ACTION ACT_AXIS:
MC_POWER(
	Axis:=REF , 
	Enable:=power_do , 
	Enable_Positive:=TRUE , 
	Enable_Negative:=TRUE , 
	Override:= , 
	BufferMode:= , 
	Options:= , 
	Status=> , 
	Busy=> , 
	Active=> , 
	Error=> , 
	ErrorID=> );
MC_Read(
	Axis:=REF , 
	Enable:=TRUE , 
	Valid=> , 
	Busy=> , 
	Error=> , 
	ErrorID=> Axis_ErrorId, 
	ErrorStop=> , 
	Disabled=> , 
	Stopping=> , 
	StandStill=> , 
	DiscreteMotion=> , 
	ContinuousMotion=> , 
	SynchronizedMotion=> , 
	Homing=> , 
	ConstantVelocity=> , 
	Accelerating=> , 
	Decelerating=> , 
	Status=> );

MC_Stop(
	Axis:=REF , 
	Execute:=stop_do , 
	Deceleration:= , 
	Jerk:= , 
	Options:= , 
	Done=> , 
	Busy=> , 
	Active=> , 
	CommandAborted=> , 
	Error=> , 
	ErrorID=> );
	IF MC_Stop.Busy THEN 
		stop_do:=FALSE;
	END_IF
MC_Reset(
	Axis:=REF , 
	Execute:=reset_do , 
	Done=> , 
	Busy=> , 
	Error=> , 
	ErrorID=> );
	IF MC_Reset.Busy THEN 
		reset_do:=FALSE;
	END_IF
MC_SetPos(
	Axis:=REF , 
	Execute:=Initialize , 
	Position:=0 , 
	Mode:= , 
	Options:= , 
	Done=> , 
	Busy=> , 
	Error=> , 
	ErrorID=> );
mc_Torque(
	Axis:= REF, 
	Execute:=var_bTorqueCtrlExecute , 
	Relative:= , 
	Torque:=var_rTorque , 
	TorqueRamp:=var_rTorqueRamp , 
	VelocityLimitHigh:= , 
	VelocityLimitLow:= , 
	BufferMode:= , 
	Options:= , 
	InTorque=> , 
	Busy=> , 
	Active=> , 
	CommandAborted=> , 
	Error=> , 
	ErrorId=> );
    IF mc_Torque.Busy THEN 
		var_bTorqueCtrlExecute:=FALSE;
	END_IF
END_ACTION

END_FUNCTION_BLOCK

// ---- POUs/100_SubTank/FB/FB_Circulation.TcPOU
FUNCTION_BLOCK FB_Circulation
VAR_INPUT	
	BottomLevel1,BottomLevel2	:BOOL;	
	MUstate						:INT;
	setoff						:BOOL;
	set_pump_voltage1			:LREAL;
	set_pump_voltage2			:LREAL;
END_VAR
VAR_OUTPUT
	CircPumpWorking1			:BOOL;
	CircPumpWorking2			:BOOL;
	error_code					:INT;
	out_pump_voltage1			:INT;
	out_pump_voltage2			:INT;
END_VAR
VAR
	Bottom_ON_filterTon1		:TON;				//滤波
	Bottom_OFF_filterTon1		:TON;
	Bottom_filterLevel1			:BOOL;
	
	Bottom_ON_filterTon2		:TON;				//滤波
	Bottom_OFF_filterTon2		:TON;
	Bottom_filterLevel2			:BOOL;
	
	filterTime_ON				:TIME;	//接通滤波时间
	filterTime_OFF				:TIME;	//接断开滤波间
	
	ton_circ1,ton_circ2:TON;
	work_ton1,work_ton2:TON;
	circ_time_trig1,circ_time_trig2:R_TRIG;
	circ_number1,circ_number2:INT;//循坏次数
	setoff_f_trig:F_TRIG;
	step_L,step_R:INT;
	state_change_trig1,state_change_trig2:R_TRIG;
	
	EL4002_CH			:ARRAY[1..2] OF FB_WriteAnalog;
	temp_pump_voltage1  :INT;
	temp_pump_voltage2  :INT;
	
END_VAR

ACT_filter_level();
ACT_circ_L();
ACT_circ_R();

IF MUstate=MUStateEnum.swapping THEN 
	filterTime_ON:=T#0S;
	filterTime_OFF:=T#0S;
ELSE
	filterTime_ON:=T#0.5S;
	filterTime_OFF:=T#0.5S;
END_IF

(************setoff***************************)
setoff_f_trig(CLK:=setoff  , Q=> );
IF setoff_f_trig.Q THEN 
	ton_circ1(IN:=FALSE);
	work_ton1(IN:=FALSE);
	ton_circ2(IN:=FALSE);
	work_ton2(IN:=FALSE);
	circ_number1:=0;	
	circ_number2:=0;	
END_IF
(************切换到SWAP或者到idle 时，需将错误复位掉*************************** 2023.1.15 无需复位
state_change_trig1(CLK:=MUstate=MUStateEnum.swapping  , Q=> );
state_change_trig2(CLK:=MUstate=MUStateEnum.idle , Q=> );
IF  state_change_trig1.Q OR state_change_trig2.Q  THEN 
		error_code:=MUErrorEnum.no_error;
		ton_circ1(IN:=FALSE);
		work_ton1(IN:=FALSE);
		ton_circ2(IN:=FALSE);
		work_ton2(IN:=FALSE);
		step_L:=step_R:=0;
END_IF
*)
(**************PUMP  SPEED********************************)
EL4002_CH[1](
	Enable:=TRUE , 
	In:=set_pump_voltage1 , 
	AnalogOffset:= , 
	Set_MaxValue:=5 , 
	MaxValue:=10 , 
	out=>temp_pump_voltage1 );
EL4002_CH[2](
	Enable:=TRUE , 
	In:=set_pump_voltage2 , 
	AnalogOffset:= , 
	Set_MaxValue:=5 , 
	MaxValue:=10 , 
	out=>temp_pump_voltage2 );

IF CircPumpWorking1 THEN 
	out_pump_voltage1:=temp_pump_voltage1;
ELSE
	out_pump_voltage1:=0;
END_IF
IF CircPumpWorking2 THEN 
	out_pump_voltage2:=temp_pump_voltage2;
ELSE
	out_pump_voltage2:=0;
END_IF

ACTION ACT_circ_L:
CASE step_L  OF 
0://
	IF MUstate=MUStateEnum.swapping THEN 
		step_L:=10;
	ELSE
		step_L:=20;
	END_IF
10://swappingg,循坏，不会报错
	IF MUstate<>MUStateEnum.swapping THEN 
		step_L:=20;
	END_IF
	
	CircPumpWorking1:=Bottom_filterLevel1 ;
20://normal,有报错
(*When pump 3 was activate less than …x/min => Alarm 1: Check circulation Left Print Heads
When pump 6 was activate less than …x/min => Alarm 2: Check circulation Right Print Heads

When pump 3 was activate less than 1x/2min =>	Alarm 3: No Circulation through Left Print Heads
When pump 6 was activate less than 1x/2min => 	Alarm 4: No Circulation through Right Print Heads

When pump 3 runs longer than 8sec => 	Alarm 5: Runtime Error Left Circulation pump 
When pump 6 runs longer than 8sec => 	Alarm 6: Runtime Error Right Circulation Pump 

*)
	IF MUstate=MUStateEnum.swapping THEN 
		step_L:=10;
	END_IF
	
	CircPumpWorking1:=Bottom_filterLevel1 ;
	
		ton_circ1(IN:=NOT ton_circ1.Q  , PT:=T#2M , Q=> , ET=> );
		circ_time_trig1(CLK:=CircPumpWorking1 , Q=> );
		IF circ_time_trig1.Q THEN 
				circ_number1:=circ_number1+1;
		END_IF
		
	(*************error********************)
	IF ton_circ1.ET >=T#1M AND ton_circ1.ET<T#2M THEN 				
		IF circ_number1<1 THEN 
			error_code:=MUErrorEnum.alarm_circulation_left;			
		END_IF
	ELSIF ton_circ1.q THEN 		
		IF circ_number1<1 THEN 
			error_code:=MUErrorEnum.alarm_through_left;
		END_IF
		(********error跳转********)
		IF error_code<>0 THEN 
			step_L:=100;
		END_IF
		circ_number1:=0;	
	END_IF
	
	work_ton1(IN:=CircPumpWorking1 , PT:=T#8S , Q=> , ET=> );
	IF work_ton1.Q THEN 
		error_code:=MUErrorEnum.alarm_runtime_circulation_left;	
		step_L:=100;
	END_IF
			
100://error
	CircPumpWorking1:=FALSE;
	circ_number1:=0;	
	ton_circ1(IN:=FALSE);
	work_ton1(IN:=FALSE);
	step_L:=0;

END_CASE
	IF 	setoff    THEN 
		error_code:=MUErrorEnum.no_error;
		step_L:=0;
	END_IF
END_ACTION

ACTION ACT_circ_R:
CASE step_R  OF 
0://
	IF MUstate=MUStateEnum.swapping THEN 
		step_R:=10;
	ELSE
		step_R:=20;
	END_IF
10://swappingg,循坏，不会报错
	IF MUstate<>MUStateEnum.swapping THEN 
		step_R:=20;
	END_IF
	
	CircPumpWorking2:=Bottom_filterLevel2 ;
20://normal,有报错
(*When pump 3 was activate less than …x/min => Alarm 1: Check circulation Left Print Heads
When pump 6 was activate less than …x/min => Alarm 2: Check circulation Right Print Heads

When pump 3 was activate less than 1x/2min =>	Alarm 3: No Circulation through Left Print Heads
When pump 6 was activate less than 1x/2min => 	Alarm 4: No Circulation through Right Print Heads

When pump 3 runs longer than 8sec => 	Alarm 5: Runtime Error Left Circulation pump 
When pump 6 runs longer than 8sec => 	Alarm 6: Runtime Error Right Circulation Pump 

*)
	IF MUstate=MUStateEnum.swapping THEN 
		step_R:=10;
	END_IF
	
	CircPumpWorking2:=Bottom_filterLevel2 ;
	
		ton_circ2(IN:=NOT ton_circ2.Q  , PT:=T#2M , Q=> , ET=> );
		circ_time_trig2(CLK:=CircPumpWorking2 , Q=> );
		IF circ_time_trig2.Q THEN 
				circ_number2:=circ_number2+1;
		END_IF
		
	(*************error********************)
	IF ton_circ2.ET >=T#1M AND ton_circ2.ET<T#2M THEN 				
		IF circ_number2<1 THEN 
			error_code:=MUErrorEnum.alarm_circulation_right;
		END_IF
	ELSIF ton_circ2.q THEN 
		IF circ_number2<1 THEN 
			error_code:=MUErrorEnum.alarm_through_right;
		END_IF
		(********error跳转********)
		IF error_code<>0 THEN 
			step_R:=100;
		END_IF
		circ_number2:=0;	
	END_IF
	
	work_ton2(IN:=CircPumpWorking2 , PT:=T#8S , Q=> , ET=> );
	IF work_ton2.Q THEN 
		error_code:=MUErrorEnum.alarm_runtime_circulation_right;
		step_R:=100;
	END_IF
				
100://error
	CircPumpWorking2:=FALSE;
	circ_number2:=0;	
	ton_circ2(IN:=FALSE);
	work_ton2(IN:=FALSE);
	step_R:=0;

	
END_CASE
	IF setoff   THEN 
		error_code:=MUErrorEnum.no_error;
		step_R:=0;
	END_IF
END_ACTION

ACTION ACT_filter_level:
(************LEVEL_BOT1*****************)
Bottom_ON_filterTon1(IN:=BottomLevel1 , PT:=filterTime_ON , Q=> , ET=> );
Bottom_OFF_filterTon1(IN:=NOT BottomLevel1 , PT:=filterTime_OFF , Q=> , ET=> );

IF Bottom_ON_filterTon1 .Q  THEN 
	Bottom_filterLevel1:=TRUE;
ELSIF Bottom_OFF_filterTon1 .Q THEN 
	Bottom_filterLevel1:=FALSE;
END_IF


(************LEVEL_BOT2*****************)
Bottom_ON_filterTon2(IN:=BottomLevel2 , PT:=filterTime_ON , Q=> , ET=> );
Bottom_OFF_filterTon2(IN:=NOT BottomLevel2 , PT:=filterTime_OFF , Q=> , ET=> );

IF Bottom_ON_filterTon2 .Q  THEN 
	Bottom_filterLevel2:=TRUE;
ELSIF Bottom_OFF_filterTon2 .Q THEN 
	Bottom_filterLevel2:=FALSE;
END_IF
END_ACTION

END_FUNCTION_BLOCK

// ---- POUs/100_SubTank/FB/FB_SubTank_C.TcPOU
FUNCTION_BLOCK FB_SubTank_C
VAR_INPUT	
	sublevel					:BOOL;
	protectLevel				:BOOL;	
	filterTime_ON				:TIME;	//接通滤波时间
	filterTime_OFF				:TIME;	//接断开滤波间
	inkFillTimeOutSet			:TIME;   //供墨超时时间设定 s	
END_VAR
VAR_OUTPUT	
	PumpWorking 				:BOOL;	//输出
	state								:INT;
	error_code					:INT;
	Error						:BOOL;
END_VAR
VAR	
	step						:INT;
	ON_filterTon			:TON;						//滤波
	OFF_filterTon			:TON;
	ON_filterTon_P			:TON;						//保护气瓶滤波
	OFF_filterTon_P			:TON;
	filterLevel			    :BOOL;
	filterLevel_P			:BOOL;
	inkFillTimeOutTon		:TON;	
END_VAR
VAR_IN_OUT
	setoff					:BOOL;
END_VAR

ACT_filter_level();

CASE step OF
0://ready
	state:=SubTankStateEnum.ready;
	(************Pumping*****************)
	IF NOT filterLevel AND NOT filterLevel_P  THEN 		
		PumpWorking :=TRUE;
	END_IF	
	IF 	 filterLevel OR  filterLevel_P  THEN
		PumpWorking :=FALSE;
	END_IF
	
	(************inkFillTimeOut*****************)
	inkFillTimeOutTon(IN:=PumpWorking   , PT:=inkFillTimeOutSet , Q=> , ET=> );
		IF inkFillTimeOutTon.Q THEN 
			error_code:=SubTankErrorEnum.pump_timeout;
			step:=100;	
		END_IF	
	
90://setoff
	error:=FALSE;	
	error_code:=ISSErrorEnum.no_error;
		
	inkFillTimeOutTon(IN:=FALSE);
	PumpWorking  :=FALSE;		
	step:=0;		
	
100://error
	state:=SubTankStateEnum.error;
	inkFillTimeOutTon(IN:=FALSE);
	PumpWorking  :=FALSE;	
	error:=TRUE;
END_CASE

IF setoff OR GVL.Reset THEN 
	setoff:=FALSE;
	step:=90;
END_IF
(*****************************************************)
	IF GVL.Emstop_Button  THEN 
		error_code:=ISSErrorEnum.emergency_error;
		step:=100;
	ELSIF filterLevel_P THEN 
		error_code:=ISSErrorEnum.back_to_air_tank;
		step:=100;
	END_IF

ACTION ACT_filter_level:
(************LEVEL*****************)
ON_filterTon(IN:=sublevel , PT:=filterTime_ON , Q=> , ET=> );
OFF_filterTon(IN:=NOT sublevel , PT:=filterTime_OFF , Q=> , ET=> );

IF ON_filterTon .Q  THEN 
	filterLevel:=TRUE;
ELSIF OFF_filterTon .Q THEN 
	filterLevel:=FALSE;
END_IF

(*************LEVEL_P****************)
ON_filterTon_P(IN:=protectLevel , PT:=filterTime_ON , Q=> , ET=> );
OFF_filterTon_P(IN:=NOT protectLevel , PT:=filterTime_OFF , Q=> , ET=> );

IF ON_filterTon_P .Q  THEN 
	filterLevel_P:=TRUE;
ELSIF OFF_filterTon_P .Q THEN 
	filterLevel_P:=FALSE;
END_IF
END_ACTION

END_FUNCTION_BLOCK

// ---- POUs/100_SubTank/FB/FB_SubTank_W.TcPOU
FUNCTION_BLOCK FB_SubTank_W
VAR_INPUT
	enable							:BOOL;
	fill_in_swap_enable				:BOOL;
	ISswappingState					:INT;//是否在换液状态
	alternate_fill					:BOOL;//交替加墨
	Toplevel          				:BOOL;
	protectLevel					:BOOL;	
	filterTime_ON					:TIME;	//接通滤波时间
	filterTime_OFF					:TIME;	//接断开滤波间
	inkFillTimeOutSet				:TIME;   //供墨超时时间设定 s	
	CircPumpWorking			        :BOOL;
END_VAR
VAR_OUTPUT	
	PumpWorking				    :BOOL;	//输出	
	state						:INT;
	error_code					:INT;
	Error						:BOOL;
END_VAR
VAR	
	step1,step2,step						:INT;
	Top_ON_filterTon				:TON;					//滤波
	Top_OFF_filterTon				:TON;
	Top_filterLevel					:BOOL;
	inkFillTimeOutTon				:TON;
	
	ON_filterTon_P			:TON;						//滤波
	OFF_filterTon_P			:TON;
	filterLevel_P				:BOOL;
	en_r_trig:R_TRIG;
	en_f_trig:F_TRIG;
	FB_SQUARE			:FB_SQUARE;
	ton1:Tc2_Standard.TON;
END_VAR
VAR_IN_OUT
	setoff					:BOOL;
END_VAR

ACT_fill();


	IF   GVL.Emstop_Button THEN 
		error_code:=ISSErrorEnum.emergency_error;
		step:=100;	
	
	ELSIF filterLevel_P THEN 
		error_code:=ISSErrorEnum.back_to_air_tank;
		step:=100;
	END_IF

ACTION ACT_fill:
ACT_filter_level();
(******************FillPumpWorking********************)
CASE step OF
0://ready
	state:=SubTankStateEnum.ready;
	
(********************供墨*************************************************************************************)	
	(************setoff*****************)	
	IF setoff OR GVL.Reset THEN 
		step:=90;
	END_IF
	IF enable THEN 
		IF ISswappingState<>MUStateEnum.swapping THEN  //正常供墨
			ACT_fill_in_normal();
		ELSE 											//交换加墨	
			ACT_fill_in_swap();
		END_IF	
	ELSE 
		inkFillTimeOutTon(IN:=FALSE);
		PumpWorking :=FALSE;
	END_IF			
90://setoff
		error:=FALSE;	
		error_code:=ISSErrorEnum.no_error;
		
		inkFillTimeOutTon(IN:=FALSE);
		PumpWorking :=FALSE;	
		step:=0;
100://error
	state:=ISSStateEnum.error;
	inkFillTimeOutTon(IN:=FALSE);
	PumpWorking :=FALSE;	
	error:=TRUE;	
END_CASE

IF setoff OR GVL.Reset THEN 
	setoff:=FALSE;
	step:=90;
END_IF
END_ACTION

ACTION ACT_fill_in_normal:
ACT_filter_level();
(******************FillPumpWorking********************)
	(************Pumping*****************)
	IF NOT filterLevel_P  AND  NOT Top_filterLevel  AND NOT CircPumpWorking THEN 
		PumpWorking:=TRUE;
	END_IF	
	IF 	 filterLevel_P  OR Top_filterLevel  OR CircPumpWorking THEN 
		PumpWorking:=FALSE;
	END_IF
	

	(************inkFillTimeOut*****************)
		inkFillTimeOutTon(IN:=PumpWorking  , PT:=inkFillTimeOutSet, Q=> , ET=> );
		IF inkFillTimeOutTon.Q THEN 
			error_code:=SubTankErrorEnum.pump_timeout;
			step:=100;	
		END_IF
END_ACTION

ACTION ACT_fill_in_swap:
en_r_trig(CLK:= fill_in_swap_enable, Q=> );
en_f_trig(CLK:=fill_in_swap_enable , Q=> );
IF en_r_trig.Q  OR en_f_trig .Q  THEN 
		PumpWorking  :=FALSE;				
		inkFillTimeOutTon(IN:=FALSE);
END_IF
(******************FillPumpWorking********************)
IF fill_in_swap_enable THEN 
		IF NOT alternate_fill THEN 
				(************all Pumping*****************)
			IF NOT filterLevel_P  AND  NOT Toplevel  AND NOT CircPumpWorking THEN 
				PumpWorking:=TRUE;
			END_IF	
			IF 	 filterLevel_P  OR Toplevel  OR CircPumpWorking THEN 
				PumpWorking:=FALSE;
			END_IF
				
			(************inkFillTimeOut*****************)
				inkFillTimeOutTon(IN:=PumpWorking  , PT:=T#2M, Q=> , ET=> );				
				IF inkFillTimeOutTon.Q THEN 
					error_code:=SubTankErrorEnum.pump_timeout;
					step:=100;			
				END_IF	
		ELSE
				(************alternate Pumping*****************)		
			IF NOT filterLevel_P  AND  NOT Toplevel  AND NOT CircPumpWorking THEN
				FB_SQUARE(T_ON:=T[2] , T_OFF:= T[3], SQUARE=> PumpWorking); 
				inkFillTimeOutTon(IN:=TRUE  , PT:=T#2M, Q=> , ET=> );
				IF inkFillTimeOutTon.Q THEN 
					error_code:=SubTankErrorEnum.pump_timeout;
					step:=100;
				END_IF
			END_IF	
			IF 	 filterLevel_P  OR Toplevel  OR CircPumpWorking THEN 
				PumpWorking:=FALSE;		
			END_IF
			
		END_IF
END_IF
END_ACTION

ACTION ACT_filter_level:
(************LEVEL_TOP*****************)
Top_ON_filterTon(IN:=Toplevel , PT:=filterTime_ON , Q=> , ET=> );
Top_OFF_filterTon(IN:=NOT Toplevel , PT:=filterTime_OFF , Q=> , ET=> );

IF Top_ON_filterTon .Q  THEN 
	Top_filterLevel:=TRUE;
ELSIF Top_OFF_filterTon .Q THEN 
	Top_filterLevel:=FALSE;
END_IF



(************LEVEL_P*****************)
ON_filterTon_P(IN:=protectLevel , PT:=filterTime_ON-T#1S , Q=> , ET=> );
OFF_filterTon_P(IN:=NOT protectLevel , PT:=filterTime_OFF-T#1S , Q=> , ET=> );

IF ON_filterTon_P .Q  THEN 
	filterLevel_P:=TRUE;
ELSIF OFF_filterTon_P .Q THEN 
	filterLevel_P:=FALSE;
END_IF
END_ACTION

END_FUNCTION_BLOCK

// ---- POUs/100_SubTank/P_SubTank.TcPOU
PROGRAM P_SubTank
VAR
	FB_SubTankFill_C   :ARRAY[1..12] OF FB_SubTank_C;
	FB_SubTankFill_P   :ARRAY[1..2] OF FB_SubTank_C;
	FB_SubTankFill_W   :ARRAY[1..2] OF FB_SubTank_W;
	FB_SubTankFill_F   :ARRAY[1..2] OF FB_SubTank_W;
	
	PumpWorking1_W,PumpWorking2_W:BOOL;
	PumpWorking1_F,PumpWorking2_F:BOOL;
	
	bqFillPumpWorking_W_r_trig:Tc2_Standard.R_TRIG;//白墨泵启动
	bqFillPumpWorking_F_r_trig:Tc2_Standard.R_TRIG;	//	清洗液泵启动
	
	i:INT;
(****************白墨循坏*******************************)
	FB_Circulation:FB_Circulation;
	
	enable_W_rtrig:Tc2_Standard.R_TRIG;
	enable_F_rtrig:Tc2_Standard.R_TRIG;
END_VAR

VAR PERSISTENT
	SubTankFill_en:ARRAY[1..4] OF BOOL:=[1,1,0,0];//w1,w2,f1,f2  白，清洗液供墨使能
END_VAR

ACT_Color();
ACT_W_F();
ACT_Circulation();
(****white pump**************************************)
stOutput.bqFillPumpWorking[13]:=(PumpWorking1_W ) 
						AND NOT stOutput.bqFillPumpWorking[19] ;
stOutput.bqFillPumpWorking[15]:=(PumpWorking2_W ) 
						AND NOT stOutput.bqFillPumpWorking[20];
(****flush pump**************************************)
stOutput.bqFillPumpWorking[19]:=(PumpWorking1_F ) 
						AND NOT stOutput.bqFillPumpWorking[13] ;
stOutput.bqFillPumpWorking[20]:=(PumpWorking2_F ) 
						AND NOT stOutput.bqFillPumpWorking[15] ;
													
(**********************墨盒里 
		0” circuit not filled (default setting)
	“1” circuit filled with “white ink”
	“2” circuit filled with “storage fluid”
******************************************************)
bqFillPumpWorking_W_r_trig(CLK:=stOutput.bqFillPumpWorking[13] OR stOutput.bqFillPumpWorking[15] , Q=> );
bqFillPumpWorking_F_r_trig(CLK:=stOutput.bqFillPumpWorking[19] OR stOutput.bqFillPumpWorking[20] , Q=> );
IF bqFillPumpWorking_W_r_trig.Q THEN
	SubTankInk_type:=1; 
ELSIF bqFillPumpWorking_F_r_trig.Q THEN 
	SubTankInk_type:=2;
END_IF


(***************切换墨水**************************)
enable_F_rtrig(CLK:= GVL_API.stMU.state=MUStateEnum.swapping AND GVL_API.stMU.cycle=0 , Q=> );
enable_W_rtrig(CLK:=GVL_API.stMU.state=MUStateEnum.swapping AND GVL_API.stMU.cycle=1 , Q=> );
IF enable_W_rtrig.Q THEN  //WHITE
	SubTankFill_en[1]:=TRUE;
	SubTankFill_en[2]:=TRUE;
	SubTankFill_en[3]:=FALSE;
	SubTankFill_en[4]:=FALSE;
ELSIF enable_F_rtrig.Q THEN //FLUSH
	SubTankFill_en[1]:=FALSE;
	SubTankFill_en[2]:=FALSE;
	SubTankFill_en[3]:=TRUE;
	SubTankFill_en[4]:=TRUE;
END_IF

ACTION ACT_Circulation:
FB_Circulation(
	BottomLevel1:=GVL.inklevel_W_L_BOT , 
	BottomLevel2:=GVL.inklevel_W_R_BOT , 
	MUstate:=GVL_API.stMU.state , 
	setoff:= GVL_API.stMU.SetOff OR GVL.Reset, 
	set_pump_voltage1:=HMI_CircPump1_V , 
	set_pump_voltage2:=HMI_CircPump2_V , 
	CircPumpWorking1=>stOutput.bqSubCircPumpWorking[1]  , 
	CircPumpWorking2=> stOutput.bqSubCircPumpWorking[2] , 
	error_code=> ,
	out_pump_voltage1=>EL4002_S[1] , 
	out_pump_voltage2=>EL4002_S[2] );
END_ACTION

ACTION ACT_Color:
(*******************COLOR***************************)
(*
1	:	LC1		2	:	LC2
3	:	LM1		4	:	LM2
5	:	Y1		6	:	Y2
7	:	M1		8	:	M2
9	:	C1		10	:	C2
11	:	K1		12	:	K2
13		P1		14		P2
15		W_L		16		W_R

*)
FOR i:=1 TO 12 DO 
	FB_SubTankFill_C[i](
		sublevel:= stInput.biSubInkTankLevel[i], 
		protectLevel:= stInput.biProtectAirTankLevel_C, 
		filterTime_ON:= T#0S, 
		filterTime_OFF:= T#3S, 
		inkFillTimeOutSet:= LREAL_TO_TIME(GVL_API.stSubTank[i].timeout) ,
		PumpWorking=> stOutput.bqFillPumpWorking[i], 
		state=> GVL_API.stSubTank[i].state, 
		error_code=> GVL_API.stSubTank[i].error_code, 
		Error=> GVL_API.stSubTank[i].Error, 
		setoff:=GVL_API.stSubTank[i].Setoff );
END_FOR

(*******************Primer***************************)
	FB_SubTankFill_P[1](
		sublevel:= stInput.biSubInkTankLevel[17], 
		protectLevel:= stInput.biProtectAirTankLevel_W, 
		filterTime_ON:= T#0S, 
		filterTime_OFF:= T#3S, 
		inkFillTimeOutSet:= LREAL_TO_TIME(GVL_API.stSubTank[13].timeout), 
		PumpWorking=> stOutput.bqFillPumpWorking[17], 
		state=> GVL_API.stSubTank[13].state, 
		error_code=> GVL_API.stSubTank[13].error_code, 
		Error=> GVL_API.stSubTank[13].Error, 
		setoff:=GVL_API.stSubTank[13].Setoff );
	FB_SubTankFill_P[2](
		sublevel:= stInput.biSubInkTankLevel[18], 
		protectLevel:= stInput.biProtectAirTankLevel_W, 
		filterTime_ON:= T#0S, 
		filterTime_OFF:= T#3S, 
		inkFillTimeOutSet:= LREAL_TO_TIME(GVL_API.stSubTank[14].timeout), 
		PumpWorking=> stOutput.bqFillPumpWorking[18], 
		state=> GVL_API.stSubTank[14].state, 
		error_code=> GVL_API.stSubTank[14].error_code, 
		Error=> GVL_API.stSubTank[14].Error, 
		setoff:=GVL_API.stSubTank[14].Setoff );
END_ACTION

ACTION ACT_W_F:
(*******************WHITE/FLUSH***************************)	
GVL.inklevel_W_L_BOT:=stInput.biSubInkTankLevel[13] ;	//W_L_BOT
GVL.inklevel_W_L_TOP:=stInput.biSubInkTankLevel[14] ;	//W_L_TOP
GVL.inklevel_W_R_TOP:=stInput.biSubInkTankLevel[15] ;	//W_R_TOP
GVL.inklevel_W_R_BOT:=stInput.biSubInkTankLevel[16] ;	//W_R_BOT


(*******************white***************************)
	FB_SubTankFill_W[1](
		enable:=SubTankFill_en[1],
		fill_in_swap_enable:=GVL.fill_W_in_swap_enable , 
		ISswappingState:=GVL_API.stMU.state  , 
		alternate_fill:= P_MaintenanceUnit.FB_Auto_Cycles_Swap.alternate_Pumping, 
		Toplevel:= GVL.inklevel_W_L_TOP, 
		protectLevel:= stInput.biProtectAirTankLevel_W, 
		filterTime_ON:= T#0S, 
		filterTime_OFF:= T#3S, 
		inkFillTimeOutSet:= inkFillTimeOutSet, 
		CircPumpWorking:= stOutput.bqSubCircPumpWorking[1], 
		PumpWorking=> PumpWorking1_W, 
		state=> GVL_API.stSubTank[15].state, 
		error_code=> GVL_API.stSubTank[15].error_code, 
		Error=> GVL_API.stSubTank[15].Error, 
		setoff:= GVL_API.stSubTank[15].Setoff);
	FB_SubTankFill_W[2](
		enable:=SubTankFill_en[2],
		fill_in_swap_enable:=GVL.fill_W_in_swap_enable , 
		ISswappingState:=GVL_API.stMU.state  , 
		alternate_fill:= P_MaintenanceUnit.FB_Auto_Cycles_Swap.alternate_Pumping, 
		Toplevel:= GVL.inkLevel_W_R_TOP, 
		protectLevel:= stInput.biProtectAirTankLevel_W, 
		filterTime_ON:= T#0S, 
		filterTime_OFF:= T#3S, 
		inkFillTimeOutSet:= inkFillTimeOutSet, 
		CircPumpWorking:= stOutput.bqSubCircPumpWorking[2], 
		PumpWorking=> PumpWorking2_W, 
		state=> GVL_API.stSubTank[16].state, 
		error_code=> GVL_API.stSubTank[16].error_code, 
		Error=> GVL_API.stSubTank[16].Error, 
		setoff:= GVL_API.stSubTank[16].Setoff);	
		
(*******************FLUSH***************************)
	FB_SubTankFill_F[1](
		enable:=SubTankFill_en[3],
		fill_in_swap_enable:=GVL.fill_F_in_swap_enable , 
		ISswappingState:=GVL_API.stMU.state  , 
		alternate_fill:= P_MaintenanceUnit.FB_Auto_Cycles_Swap.alternate_Pumping, 
		Toplevel:= GVL.inklevel_W_L_TOP, 
		protectLevel:= stInput.biProtectAirTankLevel_W, 
		filterTime_ON:= T#0S, 
		filterTime_OFF:= T#3S, 
		inkFillTimeOutSet:= inkFillTimeOutSet, 
		CircPumpWorking:= stOutput.bqSubCircPumpWorking[1], 
		PumpWorking=> PumpWorking1_F, 
		state=> GVL_API.stSubTank[15].state, 
		error_code=> GVL_API.stSubTank[15].error_code, 
		Error=> GVL_API.stSubTank[15].Error, 
		setoff:= GVL_API.stSubTank[15].Setoff);
	FB_SubTankFill_F[2](
		enable:=SubTankFill_en[4],
		fill_in_swap_enable:=GVL.fill_F_in_swap_enable , 
		ISswappingState:=GVL_API.stMU.state  , 
		alternate_fill:= P_MaintenanceUnit.FB_Auto_Cycles_Swap.alternate_Pumping, 
		Toplevel:= GVL.inkLevel_W_R_TOP, 
		protectLevel:= stInput.biProtectAirTankLevel_W, 
		filterTime_ON:= T#0S, 
		filterTime_OFF:= T#3S, 
		inkFillTimeOutSet:= inkFillTimeOutSet, 
		CircPumpWorking:= stOutput.bqSubCircPumpWorking[2], 
		PumpWorking=> PumpWorking2_F, 
		state=> GVL_API.stSubTank[16].state, 
		error_code=> GVL_API.stSubTank[16].error_code, 
		Error=> GVL_API.stSubTank[16].Error, 
		setoff:= GVL_API.stSubTank[16].Setoff);
END_ACTION

END_PROGRAM

// ---- POUs/999_TwinSAFE/P_TwinSAFE.TcPOU
PROGRAM P_TwinSAFE
VAR
	Err_Ack		AT%Q* 	:BOOL;//当出现了通讯报错时，用来做安全应答
	//Run_Stop	AT%Q* 	:BOOL;//启动或停止安全程序运行
	//Restart		AT%Q* 	:BOOL;//重启安全程序
	//Relyback	AT%Q* 	:ARRAY [1..4] OF BOOL;
	
	Com_err		AT%I* 	:BOOL;//用来显示通讯报错
	FB_err		AT%I* 	:BOOL;//用来显示功能块报错
	//FB_run		AT%I* 	:BOOL;
	
(**************FB监控**********************)	
	TwinSAFE_Group_State     					AT%I*    :USINT;
	TwinSAFE_FBstop1_State	 					AT%I*    :USINT;	
	TwinSAFE_Group_State_Enum				:TwinSAFE_Group_State_Enum;
	TwinSAFE_FB_ESTOP_State_Enum			:TwinSAFE_FB_ESTOP_State_Enum;	
	FB_COE_READ									:ARRAY[1..4] OF Tc2_EtherCAT.FB_EcCoESdoRead;
	bCoe_read											:BOOL;
	
(*************接入EL1094***********************)	
	bishuttle_crash_detector_left					:BOOL;
	bishuttle_crash_detector_right					:BOOL;
	btEmergency_stop									:BOOL;
	Emergency_stop_2904									:BOOL;
	biinterlock 			  								:ARRAY[1..8] OF BOOL;
	rely_back  												:ARRAY[1..4] OF BOOL;
	btReset													:BOOL;
	
(*******************LOG*****************)
	i:INT;
	Coe_Read_ton:ton;	
	log_ID:INT;
	last_group_state_ton:Tc2_Standard.TON;
	last_group_state:USINT;
	last_FBstop1_state_ton:Tc2_Standard.TON;
	last_FBstop1_state:USINT;
	
END_VAR

(*
EDM 接收反馈，假如多个的话，反馈用1904 ，可以用FB_ADD，此模块只可以用安全模块输入
不用1904，反馈需在PLC内，就做好合并，以一个值直接传输到TianSAFE 内的变量
*)

ACT_LOG();
ACT_Match();
stInput.btReset:=btReset;
Err_Ack:=stInput.btReset;


Coe_Read_ton(IN:=NOT Coe_Read_ton.Q  , PT:= , Q=> , ET=> );
IF Coe_Read_ton.Q THEN 
	bCoe_read:=NOT bCoe_read;
END_IF
FOR i:=1 TO 4 DO
FB_COE_READ[i](
	sNetId:= '192.168.1.138.2.1'(*'5.88.78.180.2.1'*) , 
	nSlaveAddr:=1014 , 
	nSubIndex:= INT_TO_BYTE(i), 
	nIndex:=16#7001 , 
	pDstBuf:=ADR(EL2904[1,i]) , 
	cbBufLen:=SIZEOF(EL2904[1,i]) , 
	bExecute:= bCoe_read, 
	tTimeout:= , 
	bBusy=> , 
	bError=> , 
	nErrId=> , 
	cbRead=> );
END_FOR

ACTION ACT_LOG:
(*************************LOG*******************************************)
//只记录错误
log_ID:=460;

//Com_err
AlarmActionArray[log_ID+1].AlarmMsg.EN	:=	'TwinSAFE Com_err ';
fbSetAlarm[log_ID+1](
	InUse:=TRUE , 
	//EventId:=log_ID+2 , 
	EventActive:=Com_err , 
	EventClass:=Alm_EventClass.Alarm , 
	ToTheLogFile:=TRUE, 
	ToTheHistory:=TRUE , 
 );
 
 //FB_err
AlarmActionArray[log_ID+2].AlarmMsg.EN	:=	'TwinSAFE FB_err ';
fbSetAlarm[log_ID+2](
	InUse:=TRUE , 
	//EventId:=log_ID+2 , 
	EventActive:=FB_err , 
	EventClass:=Alm_EventClass.Alarm , 
	ToTheLogFile:=TRUE, 
	ToTheHistory:=TRUE , 
 );

  //Restart
AlarmActionArray[log_ID+3].AlarmMsg.EN	:=	'TwinSAFE Restart ';
fbSetAlarm[log_ID+3](
	InUse:=TRUE , 
	//EventId:=log_ID+3 , 
	EventActive:=gvl.Reset , 
	EventClass:=Alm_EventClass.Event , 
	ToTheLogFile:=TRUE, 
	ToTheHistory:=TRUE , 
 );
 
//	TwinSAFE_Group_State
last_group_state_ton(IN:=NOT last_group_state_ton.Q  , PT:=T#200MS , Q=> , ET=> );
IF last_group_state_ton.Q THEN 
	last_group_state:=TwinSAFE_Group_State;
END_IF
CASE TwinSAFE_Group_State OF
1	:	TwinSAFE_Group_State_Enum	:=	1	;
2	:	TwinSAFE_Group_State_Enum	:=	2	;
4	:	TwinSAFE_Group_State_Enum	:=	4	;
5	:	TwinSAFE_Group_State_Enum	:=	5	;
6	:	TwinSAFE_Group_State_Enum	:=	6	;
7	:	TwinSAFE_Group_State_Enum	:=	7	;
16	:	TwinSAFE_Group_State_Enum	:=	16	;
17	:	TwinSAFE_Group_State_Enum	:=	17	;
END_CASE
AlarmActionArray[log_ID+4].AlarmMsg.EN	:=	CONCAT('TwinSAFE_Group_State:',
																	TO_STRING(TwinSAFE_Group_State_Enum));

fbSetAlarm[log_ID+4](
	InUse:=TRUE , 
	//EventId:=log_ID+2 , 
	EventActive:=last_group_state<>TwinSAFE_Group_State , 
	EventClass:=Alm_EventClass.Message , 
	ToTheLogFile:=TRUE, 
	ToTheHistory:=TRUE , 
 );

//TwinSAFE_FBstop1_State
last_FBstop1_state_ton(IN:=NOT last_FBstop1_state_ton.Q  , PT:=T#200MS , Q=> , ET=> );
IF last_FBstop1_state_ton.Q THEN 
	last_FBstop1_state:=TwinSAFE_FBstop1_State;
END_IF

CASE TwinSAFE_FBstop1_State OF
0	:	TwinSAFE_FB_ESTOP_State_Enum	:=	0	;
1	:	TwinSAFE_FB_ESTOP_State_Enum	:=	1	;
2	:	TwinSAFE_FB_ESTOP_State_Enum	:=	2	;
3	:	TwinSAFE_FB_ESTOP_State_Enum	:=	3	;
4	:	TwinSAFE_FB_ESTOP_State_Enum	:=	4	;
5	:	TwinSAFE_FB_ESTOP_State_Enum	:=	5	;
6	:	TwinSAFE_FB_ESTOP_State_Enum	:=	6	;
8	:	TwinSAFE_FB_ESTOP_State_Enum	:=	8	;
END_CASE
AlarmActionArray[log_ID+5].AlarmMsg.EN	:=	CONCAT('TwinSAFE_FBstop1_State:',
																	TO_STRING(TwinSAFE_FB_ESTOP_State_Enum));

fbSetAlarm[log_ID+5](
	InUse:=TRUE , 
	//EventId:=log_ID+2 , 
	EventActive:=last_FBstop1_state<>TwinSAFE_FBstop1_State , 
	EventClass:=Alm_EventClass.Message , 
	ToTheLogFile:=TRUE, 
	ToTheHistory:=TRUE , 
 );
END_ACTION

ACTION ACT_Match:
Emergency_stop_2904						:=(NOT EL2904[1,1] OR NOT EL2904[1,2])  ;
btEmergency_stop					:=NOT EL1904_M[1,1] OR NOT EL1904_M[1,2];

Axis[FastScan].IO.snLimitN			:=EL1904_M[1,3];
Axis[FastScan].IO.snLimitP			:=EL1904_M[1,4];
bishuttle_crash_detector_left		:=EL1904_M[2,1];
bishuttle_crash_detector_right		:=EL1904_M[2,2];
biinterlock[1]								:=EL1904_M[2,3];
biinterlock[2]								:=EL1904_M[2,4];
biinterlock[3]								:=EL1904_M[3,1];
biinterlock[4]								:=EL1904_M[3,2];
biinterlock[5]								:=EL1904_M[3,3];
biinterlock[6]								:=EL1904_M[3,4];
biinterlock[7]								:=EL1904_M[4,1];
biinterlock[8]								:=EL1904_M[4,2];
btReset										:=EL1904_M[4,3];

rely_back[1]								:=EL1904_M[5,1];
rely_back[2]								:=EL1904_M[5,2];
rely_back[3]								:=EL1904_M[5,3];
rely_back[4]								:=EL1904_M[5,4];
END_ACTION

END_PROGRAM

// ---- POUs/040_System/SystemEnvironment/P_SystemEnvironment.TcPOU
PROGRAM P_SystemEnvironment
VAR
	FB_SystemEnvironment:FB_SystemEnvironment;
	i:INT;
	log_ErrorEnum:EnvironmentErrorEnum;
	log_ID:INT;
END_VAR

ACT_LOG();
FB_SystemEnvironment(
	IO_Error:=P_Modbus_RTU.station_error[3] , 
	duration:= GVL_API.stSystemEnvironment.duration, 
	period:=GVL_API.stSystemEnvironment.period , 
	temp_measured=>GVL_API.stSystemEnvironment.temp_measured, 
	humidity_measured=> GVL_API.stSystemEnvironment.humidity_measured, 
	bqbuzzer=>stOutput.bqBuzzer , 
	Error=> GVL_API.stSystemEnvironment.Error, 
	error_code:= GVL_API.stSystemEnvironment.error_code, 
	state:= GVL_API.stSystemEnvironment.state, 
	Reset:=GVL_API.stSystemEnvironment.Reset  ,
	BuzzerOn:=GVL_API.stSystemEnvironment.BuzzerOn,
	BuzzerOff:=GVL_API.stSystemEnvironment.BuzzerOff );

ACTION ACT_LOG:
(*************************LOG*******************************************)
log_ID:=450;

//ERROR,log_ErrorEnum只能等于一个常数,   
CASE GVL_API.stSystemEnvironment.error_code  OF
0	:	log_ErrorEnum	:=	0	;
1	:	log_ErrorEnum	:=	1	;
2	:	log_ErrorEnum	:=	2	;
3	:	log_ErrorEnum	:=	3	;
4	:	log_ErrorEnum	:=	4	;
666	:	log_ErrorEnum	:=	666	;

END_CASE

AlarmActionArray[log_ID+1].AlarmMsg.EN	:=CONCAT('SystemEnvironment Error: ',TO_STRING(log_ErrorEnum));
fbSetAlarm[log_ID+1](
	InUse:=TRUE , 
	EventId:=log_ID+1 , 
	EventActive:=GVL_API.stSystemEnvironment.error_code<>0  AND GVL_API.stSystemEnvironment.error_code<>666, 
	EventClass:=Alm_EventClass.Alarm , 
	ToTheLogFile:=TRUE, 
	ToTheHistory:=TRUE , 
 );
 
//reset
AlarmActionArray[log_ID+2].AlarmMsg.EN	:=	'SystemEnvironment Reset ';
fbSetAlarm[log_ID+2](
	InUse:=TRUE , 
	EventId:=log_ID+2 , 
	EventActive:=GVL_API.stSystemEnvironment.Reset  , 
	EventClass:=Alm_EventClass.Event , 
	ToTheLogFile:=TRUE, 
	ToTheHistory:=TRUE , 
 );
 
 //buzz on
AlarmActionArray[log_ID+3].AlarmMsg.EN	:=CONCAT(('SystemEnvironment BuzzerOn duration: '),
																	LREAL_TO_STRING(GVL_API.stSystemEnvironment.duration));																	
AlarmActionArray[log_ID+3].AlarmMsg.EN	:=CONCAT(AlarmActionArray[log_ID+3].AlarmMsg.EN,', period: ');
AlarmActionArray[log_ID+3].AlarmMsg.EN	:=CONCAT(AlarmActionArray[log_ID+3].AlarmMsg.EN,
																	LREAL_TO_STRING(GVL_API.stSystemEnvironment.period));																															
fbSetAlarm[log_ID+3](
	InUse:=TRUE , 
	EventId:=log_ID+3 , 
	EventActive:=GVL_API.stSystemEnvironment.BuzzerOn  , 
	EventClass:=Alm_EventClass.Event , 
	ToTheLogFile:=TRUE, 
	ToTheHistory:=TRUE , 
 );
 
  //buzz off
AlarmActionArray[log_ID+4].AlarmMsg.EN	:='SystemEnvironment BuzzerOff ';
																													
fbSetAlarm[log_ID+4](
	InUse:=TRUE , 
	EventId:=log_ID+4 , 
	EventActive:= GVL_API.stSystemEnvironment.BuzzerOff  , 
	EventClass:=Alm_EventClass.Event , 
	ToTheLogFile:=TRUE, 
	ToTheHistory:=TRUE , 
 );
END_ACTION

END_PROGRAM

// ---- POUs/090MaintenanceUnit/FB/FB_drip_purge.TcPOU
(*不管什么时候，V7先断，再断V8,V9*)
FUNCTION_BLOCK FB_drip_purge
VAR_INPUT
	start_exe					    :BOOL;
	IntervalTime_W 			:LREAL;//min
	DripTime_W 				:LREAL;//sec
	PurgeTime_W 			:LREAL;//sec
	IntervalTime_C 			:LREAL;//min
	DripTime_C 				:LREAL;//sec
	PurgeTime_C 			   :LREAL;//sec
END_VAR
VAR_OUTPUT
	PurgeValve7				:BOOL;
	VacWhiteValve8			:BOOL;
	VacColorValve9			:BOOL;
	
END_VAR
VAR_IN_OUT
	has_dripped				:BOOL;
END_VAR
VAR
	start_r_trig:R_TRIG;
	start_f_trig:F_TRIG;
	step_change_trig:ARRAY[1..3] OF R_TRIG;
	step_change_en:BOOL;
	enable: BOOL;
	step:INT;
	step_W,step_C:INT;
	

	ton_IntervalTime_W 			:TON;//min
	ton_DripTime_W 				:TON;//sec
	ton_PurgeTime_W 			:TON;//sec
	ton_IntervalTime_C 			:TON;//min
	ton_DripTime_C 				:TON;//sec
	ton_PurgeTime_C 			:TON;//sec
	ton_delay					:TON;
	max_IntervalTime			:LREAL;
	ton_IntervalTime		 	:TON;//min
	
	Need_D_P_White:BOOL;//白墨时间到，需要滴压墨
	Need_D_P_Color:BOOL;//彩墨时间到，需要滴压墨
	step_both:INT;
	
	Dripping_trig:R_TRIG;
END_VAR

start_r_trig(CLK:= start_exe , Q=> );
start_f_trig(CLK:=start_exe , Q=> );

IF start_r_trig.Q THEN
	enable :=TRUE;
	//has_dripped:=FALSE;
END_IF
IF start_f_trig.Q OR GVL.Emstop_Button THEN
	enable :=FALSE;
	//has_dripped:=FALSE;
END_IF


(*切换条件：1：按设置时间；
2:V7,V8,V9停止时
*)
IF NOT PurgeValve7 AND NOT VacWhiteValve8 AND NOT VacColorValve9 THEN 
	step_change_en:=TRUE;
ELSE step_change_en:=FALSE;
END_IF

IF step_change_en THEN 
	IF PurgeTime_W=0  AND PurgeTime_C=0 THEN 
			step:=1;
	ELSIF DripTime_W=0 AND DripTime_C=0 AND PurgeTime_W= PurgeTime_C 
			AND IntervalTime_W=IntervalTime_C THEN 
			step:=2;
	ELSE 
			step:=3;
	END_IF
END_IF
		
CASE step OF
1:ACT_eg1();
2:ACT_eg2();
3:ACT_eg3();
END_CASE

(*Going off means the upper SW is closed
- As soon as the upper SW is restarted we read that value (is should be true if you have dripped)
- Then we  will reset that value en everything restarts all over again
*)
Dripping_trig(CLK:=PurgeValve7 OR VacWhiteValve8 OR VacColorValve9 , Q=> );
IF Dripping_trig.Q THEN 
	has_dripped:=TRUE;
END_IF

ACTION ACT_eg1:
IF enable THEN 
	ton_IntervalTime_W(IN:=NOT ton_IntervalTime_W.Q , PT:=LREAL_TO_TIME(IntervalTime_W)*1000*60 , Q=> , ET=> );
	ton_IntervalTime_C(IN:=NOT ton_IntervalTime_C.Q , PT:=LREAL_TO_TIME(IntervalTime_C)*1000*60 , Q=> , ET=> );
ELSE 
	ton_IntervalTime_W(IN:=FALSE);
	ton_IntervalTime_C(IN:=FALSE);
	ton_DripTime_W(IN:=FALSE);
	ton_DripTime_C(IN:=FALSE);
	step_W:=0;
	step_C:=0;	
	VacWhiteValve8:=FALSE;
	VacColorValve9:=FALSE;
	
END_IF
(******************Drip_White*****************************)
CASE step_W OF 
0://间隔
	IF ton_IntervalTime_W.Q THEN 
		step_W:=10;
	END_IF
10:
	IF DripTime_W>0 THEN 
		step_W:=20;
	ELSE 
		step_W:=0;
	END_IF
20:
	ton_DripTime_W(IN:=TRUE , PT:=LREAL_TO_TIME(DripTime_W)*1000 , Q=> , ET=> );
	VacWhiteValve8:=TRUE;
	IF ton_DripTime_W.Q THEN 
		step_W:=30;
	END_IF
30:
	VacWhiteValve8:=FALSE;
	ton_DripTime_W(IN:=FALSE);
	step_W:=0;
END_CASE
(******************Drip_Color*****************************)
CASE step_C OF 
0:
	IF ton_IntervalTime_C.Q THEN 
		step_C:=10;
	END_IF
10:
	IF DripTime_C>0 THEN 
		step_C:=20;
	ELSE 
		step_C:=0;
	END_IF
20:
	ton_DripTime_C(IN:=TRUE , PT:=LREAL_TO_TIME(DripTime_C)*1000 , Q=> , ET=> );
	VacColorValve9:=TRUE;
	IF ton_DripTime_C.Q THEN 
		step_C:=30;
	END_IF
30:
	VacColorValve9:=FALSE;
	ton_DripTime_C(IN:=FALSE);
	step_C:=0;	
END_CASE
END_ACTION

ACTION ACT_eg2:
IF enable THEN 
	ton_IntervalTime_W(IN:=NOT ton_IntervalTime_W.Q , PT:=LREAL_TO_TIME(IntervalTime_W)*1000*60 , Q=> , ET=> );
ELSE 
	ton_IntervalTime_W(IN:=FALSE);
	ton_IntervalTime_C(IN:=FALSE);
	ton_PurgeTime_W(IN:=FALSE);
	ton_PurgeTime_C(IN:=FALSE);
END_IF
(******************purge_White/Color****************************)
CASE step_W OF 
0://间隔
	IF ton_IntervalTime_W.Q THEN 
		step_W:=10;
	END_IF
10:
	IF PurgeTime_W>0 THEN 
		step_W:=20;
	ELSE 
		step_W:=0;
	END_IF
20:(**关闭功能时，先关V7在关其他*)
	ton_PurgeTime_W(IN:=TRUE , PT:=LREAL_TO_TIME(PurgeTime_W)*1000 , Q=> , ET=> );	
	VacWhiteValve8:=TRUE;
	VacColorValve9:=TRUE;
	PurgeValve7:=TRUE;
	IF ton_PurgeTime_W.Q OR start_f_trig.Q THEN 
		step_W:=30;
	END_IF
30:
	PurgeValve7:=FALSE;	
	ton_PurgeTime_W(IN:=FALSE);
	ton_delay(IN:=TRUE, PT:=T#1S , Q=> , ET=> );
	IF ton_delay.Q  THEN 
		step_W:=40;
	END_IF
40:
	ton_delay(IN:=FALSE);
	VacWhiteValve8:=FALSE;
	VacColorValve9:=FALSE;
	step_W:=0;
END_CASE
END_ACTION

ACTION ACT_eg3:
(*1:先白墨滴;2:白墨压;3:彩墨滴;4:彩墨压;*)
max_IntervalTime:=MAX(IntervalTime_W,IntervalTime_C);
(*******单独计数，有时间差******)
IF enable THEN 
	ton_IntervalTime(IN:=NOT ton_IntervalTime.Q , PT:=LREAL_TO_TIME(max_IntervalTime)*1000*60 , Q=> , ET=> );
	ton_IntervalTime_W(IN:=NOT ton_IntervalTime_W.Q , PT:=LREAL_TO_TIME(IntervalTime_W)*1000*60 , Q=> , ET=> );
	ton_IntervalTime_C(IN:=NOT ton_IntervalTime_C.Q , PT:=LREAL_TO_TIME(IntervalTime_C)*1000*60 , Q=> , ET=> );
ELSE 
	ton_IntervalTime_W(IN:=FALSE);
	ton_IntervalTime_C(IN:=FALSE);
	ton_DripTime_W(IN:=FALSE);
	ton_DripTime_C(IN:=FALSE);
	ton_IntervalTime(IN:=FALSE);
	
	PurgeValve7:=FALSE;	
	Need_D_P_White:=FALSE;
	Need_D_P_Color:=FALSE;
	
END_IF
IF ton_IntervalTime_W.Q AND (DripTime_W>0 OR PurgeTime_W>0)  THEN 
	Need_D_P_White:=TRUE;
END_IF
IF ton_IntervalTime_C.Q AND (DripTime_C>0 OR PurgeTime_C>0)  THEN 
	Need_D_P_Color:=TRUE;
END_IF

CASE step_both OF
0://因2个计时器有时间差
	IF Need_D_P_White OR  Need_D_P_Color THEN 
		step_both:=5;
	END_IF
5://当有一个时，延迟一段时间再判断
	ton_delay(IN:=TRUE, PT:=T#500MS , Q=> , ET=> );
	IF ton_delay.Q  THEN
		ton_delay(IN:=FALSE);
		step_both:=6;		
	END_IF
6://判断
	IF Need_D_P_White THEN 
		Need_D_P_White:=FALSE;
		step_both:=10;	
	ELSIF NOT Need_D_P_White AND Need_D_P_Color THEN 
		Need_D_P_Color:=FALSE;
		step_both:=110;	
	ELSE 
		step_both:=0;	
	END_IF
(***************white***********************)
10:
	IF DripTime_W>0 THEN 
		step_both:=20;//有滴墨
	ELSE 
		step_both:=40;//无滴墨，有压墨
	END_IF
20://白滴墨
	ton_DripTime_W(IN:=TRUE , PT:=LREAL_TO_TIME(DripTime_W)*1000 , Q=> , ET=> );
	VacWhiteValve8:=TRUE;
	IF ton_DripTime_W.Q  THEN 
		step_both:=30;
	ELSIF start_f_trig.Q THEN 
		step_both:=21;
	END_IF
21://停止滴墨
	VacWhiteValve8:=FALSE;	
	Need_D_P_White:=FALSE;
	step_both:=0;
30://白滴墨结束
	ton_DripTime_W(IN:=FALSE);
	IF PurgeTime_W=0 THEN //无压墨
		VacWhiteValve8:=FALSE;
		Need_D_P_White:=FALSE;
		step_both:=100;
	ELSE
		step_both:=40;
	END_IF
40://白压墨
	ton_PurgeTime_W(IN:=TRUE , PT:=LREAL_TO_TIME(PurgeTime_W)*1000 , Q=> , ET=> );	
	VacWhiteValve8:=TRUE;
	PurgeValve7:=TRUE;
	IF ton_PurgeTime_W.Q OR start_f_trig.Q THEN 
		step_both:=50;
	END_IF
50://压墨结束
	PurgeValve7:=FALSE;	
	ton_PurgeTime_W(IN:=FALSE);
	ton_delay(IN:=TRUE, PT:=T#1S , Q=> , ET=> );
	IF ton_delay.Q  THEN 
		step_both:=60;
	END_IF
60://delay
	ton_delay(IN:=FALSE);
	VacWhiteValve8:=FALSE;
	Need_D_P_White:=FALSE;
	step_both:=100;

100://先间隔1S
	ton_delay(IN:=TRUE, PT:=T#1S , Q=> , ET=> );
	IF ton_delay.Q  THEN
		ton_delay(IN:=FALSE);
		step_both:=6;		
	END_IF
	(**************color**********************)
110:	
	IF DripTime_C>0 THEN 
		step_both:=120;//有滴墨
	ELSE 
		step_both:=140;//无滴墨，有压墨
	END_IF
120://彩滴墨
	ton_DripTime_C(IN:=TRUE , PT:=LREAL_TO_TIME(DripTime_C)*1000 , Q=> , ET=> );
	VacColorValve9:=TRUE;
	IF ton_DripTime_C.Q THEN 
		step_both:=130;
	END_IF
130://彩滴墨结束
	ton_DripTime_C(IN:=FALSE);
	IF PurgeTime_C=0 THEN 
		VacColorValve9:=FALSE;
		Need_D_P_Color:=FALSE;
		step_both:=100;
	ELSE 
		step_both:=140;
	END_IF
140://彩压墨
	ton_PurgeTime_C(IN:=TRUE , PT:=LREAL_TO_TIME(PurgeTime_C)*1000 , Q=> , ET=> );	
	VacColorValve9:=TRUE;
	PurgeValve7:=TRUE;
	IF ton_PurgeTime_C.Q OR start_f_trig.Q THEN 
		step_both:=150;
	END_IF
150:
	PurgeValve7:=FALSE;	
	ton_PurgeTime_C(IN:=FALSE);
	ton_delay(IN:=TRUE, PT:=T#1S , Q=> , ET=> );
	IF ton_delay.Q  THEN 
		step_both:=160;
	END_IF
160:
	ton_delay(IN:=FALSE);
	VacColorValve9:=FALSE;
	Need_D_P_Color:=FALSE;
	step_both:=0;
END_CASE
END_ACTION

END_FUNCTION_BLOCK

// ---- POUs/080SpitUnit/FB/FB_HomeSpitUnit.TcPOU
FUNCTION_BLOCK FB_HomeSpitUnit
(*========================================
Execute需一直有效，功能块才会一直执行
先回原点，在碰右极限,再回原点
==========================================*)
VAR_IN_OUT
	Axis				:AXIS_REF;	(* B *)
END_VAR
VAR_INPUT
	Execute						:BOOL;	(* B *)
	PosLimit					:BOOL;			(*正极限位信号*)
	Position						:LREAL			(* B *) := DEFAULT_HOME_POSITION;
	HomeingVelo				:LREAL:=5;
	Standby_position		:LREAL;		//最终待机位
	bCalibrationCam 		:BOOL;	(* V *)	(* Beckhoff proprietary input *)
	rel_dis         				:LREAL:=10;  //碰到原点后，正向移动距离，在开始寻原点
	reset							:BOOL;
	maxDistance				:LREAL;
END_VAR
VAR_OUTPUT
	Done				:BOOL;	(* B *)
	Busy				:BOOL;	(* E *)
	Active				:BOOL;	(* E *)
	CommandAborted		:BOOL;	(* E *)
	Error				:BOOL;	(* B *)
	ErrorID				:UDINT;	(* E *)
END_VAR
VAR
	mcJog			:MC_Jog;
	mcHome			:MC_Home;
	mcRel           :MC_MoveRelative;
	mcAbs           :MC_MoveAbsolute;	
	mcStop			:MC_Stop;
	HomeStep		:INT;
	ton				:TON;
	StopDo			:BOOL;
	startPos		:LREAL;
	trig_start		:Tc2_Standard.R_TRIG;
END_VAR

IF  NOT Execute THEN
	mcHome.Execute		:=FALSE;
	mcRel.Execute			:=FALSE;
	mcAbs.Execute			:=FALSE;
	done							:=FALSE;
	busy							:=FALSE;	
	HomeStep					:=0;
END_IF

IF reset THEN 
	Error					:=FALSE;
END_IF

CASE HomeStep OF

0:
	busy	:=FALSE;
	Done	:=FALSE;
	mcHome.Execute	:=FALSE;
	trig_start(CLK:=FALSE );
	startPos:=0;
	IF 	Execute AND NOT Error  THEN		
		IF  NOT bCalibrationCam THEN
			HomeStep	:=10;
		ELSE
			HomeStep	:=20;
		END_IF
		busy	:=TRUE;		
	END_IF
	
10:(*先向负限位方向运动*)
	mcJog.JogForward		:=FALSE;
	mcJog.JogBackwards		:=TRUE;	
	trig_start(CLK:=mcJog.JogForward , Q=> );
	IF trig_start .Q THEN 
		startPos:=Axis.NcToPlc.ActPos;
	END_IF
	 
	IF	bCalibrationCam THEN
		mcJog.JogBackwards	:=FALSE;
		HomeStep	:=20;
	ELSIF mcJog.Error  THEN
			HomeStep	:=100;
	ELSIF NOT bCalibrationCam AND ABS(startPos-Axis.NcToPlc.ActPos)>maxDistance THEN 
			HomeStep	:=100;
	END_IF
	
20:(*从原点处正方向移动一段距离*)
	trig_start(CLK:=FALSE );
	mcRel.Execute		:=TRUE;	
	IF mcRel.Done AND Axis.Status.NotMoving THEN 
		mcRel.Execute	:=FALSE;
		HomeStep		:=30;
	ELSIF mcRel.Error  THEN 
		HomeStep	:=100;	
	END_IF
	
	(*****正向离开原点停止***********************************
	trig_start(CLK:=FALSE );
	mcJog.JogForward		:=TRUE;
	IF	NOT bCalibrationCam THEN
		mcJog.JogForward	:=FALSE;
		HomeStep	:=30;
	ELSIF mcJog.Error  THEN
			HomeStep	:=100;
	END_IF
	*)
30:(*调用回零功能块*)
	mcHome.Execute	:=TRUE;
	IF mcHome.Done AND AXIS.Status.Homed THEN
		mcHome.Execute	:=FALSE;	
		HomeStep		:=50;
	ELSIF AXIS.Status.Error  THEN
		HomeStep		:=100;
	END_IF
50:(*回待机位*)
	mcAbs.Execute:=TRUE;
	IF mcAbs.Done AND Axis.Status.NotMoving THEN 
		mcAbs.Execute	:=FALSE;
		done			:=TRUE;
		HomeStep		:=99; 		
	END_IF	
99:
	;	

100:
	Error			:=TRUE;
	trig_start(CLK:=FALSE );
	IF	mcHome.ErrorID <> 0 THEN
		ErrorID			:=mcHome.ErrorID;
	ELSIF  mcJog.ErrorID <> 0 THEN
		ErrorID			:=mcJog.ErrorID;
	ELSIF mcRel.ErrorID<>0 THEN 
		ErrorID			:=mcRel.ErrorID;
	ELSIF mcAbs.ErrorID<>0 THEN 
		ErrorID			:=mcAbs.ErrorID;	
	END_IF
	mcJog.JogForward			:=FALSE;
	mcJog.JogBackwards		:=FALSE;	
	mcRel.Execute				:=FALSE;
	mcHome.Execute			:=FALSE;
	StopDo							:=TRUE;
	HomeStep						:=0;
	
END_CASE


Call_FB();

ACTION Call_FB:
Axis.ReadStatus();
mcJog
	(
	Velocity:=	HomeingVelo ,
	Mode:=		MC_JOGMODE_CONTINOUS ,
	Axis:=		Axis ,
	);

mcHome
	(
	Execute:= ,
	Position:=			Position ,
	HomingMode:= 		,
	BufferMode:= 		,
	Options:=			 ,
	bCalibrationCam:=	bCalibrationCam ,
	Axis:=				Axis ,
	);

mcRel(
	Axis:=Axis , 
	Execute:= , 
	Distance:=rel_dis , 
	Velocity:= HomeingVelo, 
	Acceleration:= , 
	Deceleration:= , 
	Jerk:= , 
	BufferMode:= , 
	Options:= , 
	Done=> , 
	Busy=> , 
	Active=> , 
	CommandAborted=> , 
	Error=> , 
	ErrorID=> );
mcAbs(
	Axis:=Axis , 
	Execute:= , 
	Position:=Standby_position , 
	Velocity:=HomeingVelo , 
	Acceleration:= , 
	Deceleration:= , 
	Jerk:= , 
	BufferMode:= , 
	Options:= , 
	Done=> , 
	Busy=> , 
	Active=> , 
	CommandAborted=> , 
	Error=> , 
	ErrorID=> );
mcStop(
	Axis:=Axis , 
	Execute:=StopDo , 
	Deceleration:= , 
	Jerk:= , 
	Options:= , 
	Done=> , 
	Busy=> , 
	Active=> , 
	CommandAborted=> , 
	Error=> , 
	ErrorID=> );
IF mcStop.Busy THEN 
	StopDo:=FALSE;
END_IF
END_ACTION

END_FUNCTION_BLOCK

// ---- POUs/080SpitUnit/FB/FB_MoveSpitUnit_Exte.TcPOU
FUNCTION_BLOCK FB_MoveSpitUnit_Exte
VAR_INPUT
	ref		:AXIS_REF;

	Acceleration		:LREAL;
	Deceleration		:LREAL;
	Jerk				:LREAL;
END_VAR
VAR_OUTPUT	
END_VAR
VAR
	MC_Read:MC_ReadStatus;
	MC_ABS:MC_MoveAbsolute;
	MC_stop:MC_Stop;
	
	step1,step2,step3		:INT;	
	R_TRIG1,R_TRIG2,R_TRIG3	:R_TRIG;
	R_TRIG_done				:R_TRIG;
	abs_do					:BOOL;
	stop_do					:BOOL;
	error					:BOOL;

	MoveAbsolute_Busy		:BOOL;
	FB_START_r_trig:		R_TRIG;
	start					:BOOL;
	velo					:LREAL;
END_VAR
VAR_IN_OUT 
	MoveAbsExe					:BOOL;
	Velo_up						:LREAL;	//mm/s
	Velo_down						:LREAL;	//mm/s
	TargetAbs					:LREAL;//mm						
	Done						:BOOL;
	
END_VAR

(*********************NOT MOVING TIMEOUT***************************)
FB_START_r_trig(CLK:=MoveAbsExe, Q=> );
IF FB_START_r_trig.Q THEN 
	start:=TRUE;
END_IF

Call_FB();
MoveAbsolute();

(*********************error***************************)
IF  MC_Read.Error  THEN	
	start:=FALSE;
	error:=FALSE;
	step1:=step2:=step2:=0;	
	MoveAbsExe:=FALSE;
	TargetAbs:=0;

	R_TRIG1(CLK:=FALSE);
	R_TRIG2(CLK:=FALSE);
	R_TRIG3(CLK:=FALSE);
END_IF

(*********************move done***************************)
IF MoveAbsolute_Busy  THEN 
	Done:=FALSE;
END_IF

R_TRIG_done(CLK:=MC_ABS.Done OR MC_stop.Done   , Q=> );
IF R_TRIG_done.Q THEN 	
	start:=FALSE;
	R_TRIG_done(CLK:=FALSE);
	step1:=step2:=step2:=0;	
	MoveAbsExe:=FALSE;
	TargetAbs:=0;	
	Done:=TRUE ;
END_IF

ACTION Call_FB:
MC_Read(
	Axis:=ref , 
	Enable:=TRUE);

MC_ABS(
	Axis:=ref , 
	Execute:=abs_do , 
	Position:=TargetAbs , 
	Velocity:=Velo , 
	Acceleration:=Acceleration , 
	Deceleration:=Deceleration , 
	Jerk:=Jerk , 
	BufferMode:= , 
	Options:= , 
	Done=> , 
	Busy=>MoveAbsolute_Busy , 
	Active=> , 
	CommandAborted=> , 
	Error=> , 
	ErrorID=> );
	IF MC_ABS.Busy THEN 
		abs_do:=FALSE;
		MoveAbsExe:=FALSE;
	END_IF

MC_stop(
	Axis:=ref , 
	Execute:=stop_do , 
	Deceleration:=Deceleration , 
	Jerk:=Jerk , 
	Options:= , 
	Done=> , 
	Busy=> , 
	Active=> , 
	CommandAborted=> , 
	Error=> , 
	ErrorID=> );
IF MC_stop.Done THEN 
	stop_do:=FALSE;
END_IF
END_ACTION

ACTION MoveAbsolute:
(****************ABS********************)
R_TRIG2(CLK:=MoveAbsExe AND Ref.Status.NotMoving    , Q=> );

CASE step2 OF 
	0:				
		IF R_TRIG2.Q THEN 
			R_TRIG2(CLK:=FALSE);			
			MoveAbsExe:=FALSE;

			step2:=1;
		END_IF
	1:	
		IF ref.NcToPlc.ActPos>TargetAbs THEN 
			velo:=Velo_down;
			abs_do:=TRUE;
			step2:=2;
		ELSIF ref.NcToPlc.ActPos<TargetAbs THEN 
			velo:=Velo_up;
			abs_do:=TRUE;
			step2:=2;
		END_IF

	2:
		IF MC_ABS.Busy THEN 
			abs_do:=FALSE;								
			step2 :=0;
		END_IF	
END_CASE
END_ACTION

END_FUNCTION_BLOCK

// ---- POUs/080SpitUnit/P_SpitUnit.TcPOU
PROGRAM P_SpitUnit 
VAR
	ID						:INT:=SpitUnit;
	SysStep:				DINT;	
	HomeStep:				DINT;	
	RestStep				:DINT;
	MoveStep				:DINT;
	SetoffStep				:DINT;
	HomeDone:               BOOL;
	
	ton1:Tc2_Standard.TON;
	Move_Done				:BOOL;
	FB_HomeSpitUnit				:FB_HomeSpitUnit;
	FB_Move					:FB_MoveSpitUnit_Exte;
	parameter_out_of_range	:BOOL;
	
	log_ErrorEnum:SpitUnitErrorEnum;
	log_ID:INT;
	
	ton_fan:Tc2_Standard.TON;
	R_TRIG_FAN:Tc2_Standard.R_TRIG;
	F_TRIG_FAN:Tc2_Standard.F_TRIG;
	en_ton:BOOL;
	ton_commandtimeout:Tc2_Standard.TON;
	
END_VAR

ACT_FAN();
ACT_LOG();
GVL_API.stSpitUnit.ControlLoopClosed:=Axis[ID].Ref.Status .ControlLoopClosed;
(*****************POS******************************)
GVL_API.stSpitUnit.current_position:=Axis[ID].Ref.NcToPlc.ActPos;
GVL_API.stSpitUnit.home_sensor_covered:=Axis[ID].IO.snHome;

(*****************SysStep******************************)
CASE SysStep OF
0:	(*off*)
	_00_Waiting();				
100:(*idle*)		
	_100_Idle();								
200:(*home*)		
	_200_Homing();
300:(*ready*)	
	_300_Ready();							
		
500:(*Moving*)
	_500_Moving();	
600:(*Stopping*)
700:(*Error*)
	_700_Error();	
800:
	_800_SetOff();
END_CASE
IF GVL_API.stSpitUnit.SetOff OR GVL.Reset THEN 
	SysStep:=800;	
END_IF

ACT_SAFETY();


Axis[ID].aReadStatus();
Axis[ID].aReset();

ACTION _00_Waiting:
IF GVL_API.stSpitUnit.initialize THEN 
	GVL_API.stSpitUnit.initialize:=FALSE;
	SysStep:=100;
ELSIF GVL_API.stSpitUnit.homeExe THEN 
	GVL_API.stSpitUnit.homeExe:=FALSE;  
	GVL_API.stSpitUnit.Home_Done:=FALSE;
	SysStep:=200;
ELSIF GVL_API.stSpitUnit.MoveAbsoluteExe THEN 
	GVL_API.stSpitUnit.Move_Done:=FALSE;
	SysStep:=300;	
ELSIF GVL_API.stSpitUnit.SetOff OR GVL.Reset THEN 
	SysStep:=800;	
END_IF

ton1(IN:=GVL_API.stSpitUnit.Home_Done OR  GVL_API.stSpitUnit.Move_Done , PT:=State_reset_time , Q=> , ET=> );
IF ton1.Q THEN 
	GVL_API.stSpitUnit.Home_Done:=FALSE;
	GVL_API.stSpitUnit.Move_Done:=FALSE;
END_IF
END_ACTION

ACTION _100_Idle:
Axis[ID].aPower(power_do:=TRUE);	


IF   axis[Id].Ref.Status .ControlLoopClosed THEN 
		GVL_API.stSpitUnit.state:=AxisStateEnum.idle;
ELSIF GVL.Emstop_Button OR GVL.Emstop_SAFE THEN 
	GVL_API.stSpitUnit.error_code:=SpitUnitErrorEnum.emergency_error;
		SysStep:=700;
END_IF

(*****************valid command********************)
IF GVL_API.stSpitUnit.state=AxisStateEnum.idle AND GVL_API.stSpitUnit.moving_speed_down>0 AND 
GVL_API.stSpitUnit.spindle_length>0 AND GVL_API.stSpitUnit.moving_speed_up>0  THEN
	SysStep:=200;
END_IF

(*******************commandtimeout*********************************)
ton_commandtimeout(IN:=NOT axis[Id].Ref.Status .ControlLoopClosed , 
	PT:=T#10S ,
	Q=> , ET=> );
IF ton_commandtimeout.Q  THEN 
	ton_commandtimeout(IN:=FALSE );
	GVL_API.stSpitUnit.error_code:=Axis_XY_ErrorEnum.cmd_timeout;
	SysStep:=700;	
END_IF
END_ACTION

ACTION _200_Homing:
	FB_HomeSpitUnit(
		Axis:= Axis[ID].Ref, 
		Execute:= , 
		PosLimit:= Axis[ID].IO.snLimitP, 
		Position:= 0, 
		HomeingVelo:= GVL_API.stSpitUnit.moving_speed_down, 
		Standby_position:=0 , 
		bCalibrationCam:= Axis[ID].IO.snHome, 
		rel_dis:= 1, 
		reset:= , 
		maxDistance:= GVL_API.stSpitUnit.spindle_length, 
		Done=> , 
		Busy=> , 
		Active=> , 
		CommandAborted=> , 
		Error=> , 
		ErrorID=> );
	
		
CASE HomeStep OF
0:
	IF GVL_API.stSpitUnit.moving_speed_down<>0 THEN 
		HomeStep:=10;
	END_IF
10:
	FB_HomeSpitUnit.Execute:=TRUE;					
	IF FB_HomeSpitUnit.Done THEN
		GVL_API.stSpitUnit.Home_Done:=TRUE;
		FB_HomeSpitUnit.Execute:=FALSE;
		HomeStep:=20;
	END_IF
	IF FB_HomeSpitUnit.Error THEN 
		GVL_API.stSpitUnit.error_code:=SpitUnitErrorEnum.homing_error;
		HomeStep:=30;
	END_IF
	
20:	(**********HOME DONE****************)
	GVL_API.stSpitUnit.state:=SpitUnitStateEnum.ready;
	GVL_API.stSpitUnit.Homing:=FALSE;
	HomeStep:=0;
	SysStep:=0;
30:(**********TIME OUT****************)
	FB_HomeSpitUnit.Execute:=FALSE;
	FB_HomeSpitUnit.reset:=TRUE;
	HomeStep:=40;
40:(**********RESET****************)
	FB_HomeSpitUnit.reset:=FALSE;
	HomeStep:=0;
	SysStep:=700;
		
END_CASE

IF FB_HomeSpitUnit.Busy THEN 
	GVL_API.stSpitUnit.state:=SpitUnitStateEnum.homing;
	GVL_API.stSpitUnit.Homing:=TRUE;
END_IF
END_ACTION

ACTION _300_Ready:
Axis[ID].aStop();
GVL_API.stSpitUnit.Home_Done:=FALSE;	
(***********parameter_out_of_range***********)
IF GVL_API.stSpitUnit.target_position>GVL_API.stSpitUnit.spindle_length OR GVL_API.stSpitUnit.target_position<0 THEN 
		parameter_out_of_range:=TRUE;
ELSE
		parameter_out_of_range:=FALSE;
END_IF	


(*****************state******************************)
IF Axis[ID].Ref.Status.NotMoving AND axis[Id].Ref.Status .ControlLoopClosed  
AND NOT Axis[ID].Ref.Status.Error THEN 
	IF parameter_out_of_range THEN 
		GVL_API.stSpitUnit.error_code:=SpitUnitErrorEnum.parameter_out_of_range;		
		SysStep:=700;
	ELSE
		GVL_API.stSpitUnit.state:=SpitUnitStateEnum.ready;
		GVL_API.stSpitUnit.error_code:=SpitUnitErrorEnum.no_error;
	END_IF
END_IF

(*****************valid command******************************)
IF NOT parameter_out_of_range AND axis[Id].Ref.Status .ControlLoopClosed  THEN  			
	IF GVL_API.stSpitUnit.MoveAbsoluteExe	 THEN 	
			SysStep:=500;
	ELSIF GVL_API.stSpitUnit.homeExe  THEN			
			SysStep:=200;  	  							
	END_IF
END_IF

(*****************SETOFF******************************)
IF GVL_API.stSpitUnit.setoff THEN
	 SysStep:=0;
END_IF
END_ACTION

ACTION _500_Moving:
IF Axis[ID].Ref.Status.Moving THEN 
	GVL_API.stSpitUnit.state:=SpitUnitStateEnum.moving;
END_IF


IF  GVL_API.stSpitUnit.Move_Done  THEN 			(************/Move_Done**************)			
	GVL_API.stSpitUnit.state:=SpitUnitStateEnum.ready;	
	SysStep:=0;
ELSIF Axis[ID].Ref.Status.Moving THEN 				(************trigger_limit**************)
	IF Axis[ID].Ref.Status.PositiveDirection AND Axis[ID].IO.snLimitP  
	THEN	
		Axis[ID].aStop(stop_do:=TRUE);
		GVL_API.stSpitUnit.error_code:=SpitUnitErrorEnum.trigger_limit;
		SysStep:=700;	
	END_IF 
ELSE GVL_API.stSpitUnit.error_code:=SpitUnitErrorEnum.no_error;
END_IF

IF NOT parameter_out_of_range THEN 
	FB_Move(
	ref:= Axis[ID].Ref, 
	Acceleration:= GVL_API.stSpitUnit.acceleration, 
	Deceleration:= GVL_API.stSpitUnit.acceleration, 
	Jerk:= , 
	MoveAbsExe:= GVL_API.stSpitUnit.MoveAbsoluteExe, 
	Velo_up:= GVL_API.stSpitUnit.moving_speed_up, 
	Velo_down:=GVL_API.stSpitUnit.moving_speed_down , 
	TargetAbs:= GVL_API.stSpitUnit.target_position, 
	Done:=GVL_API.stSpitUnit.Move_Done );

END_IF
END_ACTION

ACTION _700_Error:
(*****************ERROR******************************)
GVL_API.stSpitUnit.Error:=TRUE;
GVL_API.stSpitUnit.state:=SpitUnitStateEnum.error;
		GVL_API.stSpitUnit.initialize:=FALSE;
		GVL_API.stSpitUnit.homeExe:=FALSE; 
		GVL_API.stSpitUnit.MoveAbsoluteExe:=FALSE;		
		FB_HomeSpitUnit.Execute:=FALSE;
		GVL_API.stSpitUnit.Homing:=FALSE;
		GVL_API.stSpitUnit.Home_Done:=FALSE;
		GVL_API.stSpitUnit.Move_Done:=FALSE;

 SysStep:=0;
END_ACTION

ACTION _800_SetOff:
Axis[ID].aStop();
(*****************SETOFF*****************************)
CASE SetoffStep OF
0:(***************复位命令**************************)
	IF GVL_API.stSpitUnit.setoff OR GVL.Reset THEN
		GVL_API.stSpitUnit.initialize:=FALSE;
		GVL_API.stSpitUnit.homeExe:=FALSE; 
		GVL_API.stSpitUnit.MoveAbsoluteExe:=FALSE;		
		FB_HomeSpitUnit(Axis:= Axis[ID].Ref, Execute:= FALSE);
		GVL_API.stSpitUnit.Homing:=FALSE;
		GVL_API.stSpitUnit.Home_Done:=FALSE;
		GVL_API.stSpitUnit.Move_Done:=FALSE;
		SetoffStep:=1;
	END_IF
1:	
	SetoffStep:=10;
10:	(***************轴错误复位**************************)	
		parameter_out_of_range:=FALSE;		
		Axis[ID].Reset_do:=TRUE;		
		SetoffStep:=100;		
100:		
	IF Axis[ID].Ref.Status.NotMoving THEN 
		GVL_API.stSpitUnit.setoff:=FALSE;
		Axis[Id].aPower(power_do:=FALSE);
		GVL_API.stSpitUnit.Error:=FALSE;
		GVL_API.stSpitUnit.state:=SpitUnitStateEnum.off;
		GVL_API.stSpitUnit.error_code:=SpitUnitErrorEnum.no_error;
		
		SysStep:=0;
		SetoffStep:=0;
	END_IF
	  
END_CASE
END_ACTION

ACTION ACT_FAN:
R_TRIG_FAN(CLK:=GVL_API.stSpitUnit.FanState , Q=> );
F_TRIG_FAN(CLK:=GVL_API.stSpitUnit.FanState , Q=> );
IF R_TRIG_FAN.Q THEN 
	stOutput.bqFanPower:=TRUE;
END_IF


IF F_TRIG_FAN.Q THEN 
	en_ton:=TRUE;
END_IF
ton_fan(IN:= en_ton  , PT:=T#10S , Q=> , ET=> );
IF ton_fan.Q THEN 
	en_ton:=FALSE;
	stOutput.bqFanPower:=FALSE;
END_IF
END_ACTION

ACTION ACT_LOG:
(*************************LOG*******************************************)
log_ID:=580;
//initialize
AlarmActionArray[log_ID+1].AlarmMsg.EN	:=	CONCAT('SpitUnit Initialize maxDistance:',
																	LREAL_TO_STRING(GVL_API.stSpitUnit.spindle_length));
AlarmActionArray[log_ID+1].AlarmMsg.EN	:=	CONCAT(AlarmActionArray[log_ID+1].AlarmMsg.EN,'; velocity_up:');
AlarmActionArray[log_ID+1].AlarmMsg.EN	:=	CONCAT(AlarmActionArray[log_ID+1].AlarmMsg.EN,
																	LREAL_TO_STRING(GVL_API.stSpitUnit.moving_speed_up));	
AlarmActionArray[log_ID+1].AlarmMsg.EN	:=	CONCAT(AlarmActionArray[log_ID+1].AlarmMsg.EN,'; velocity_down:');	
AlarmActionArray[log_ID+1].AlarmMsg.EN	:=	CONCAT(AlarmActionArray[log_ID+1].AlarmMsg.EN,
																	LREAL_TO_STRING(GVL_API.stSpitUnit.moving_speed_down));																															
AlarmActionArray[log_ID+1].AlarmMsg.EN	:=	CONCAT(AlarmActionArray[log_ID+1].AlarmMsg.EN,'; acc:');	
AlarmActionArray[log_ID+1].AlarmMsg.EN	:=	CONCAT(AlarmActionArray[log_ID+1].AlarmMsg.EN,
																	LREAL_TO_STRING(GVL_API.stSpitUnit.acceleration));	
//AlarmActionArray[log_ID+1].AlarmMsg.EN	:=	'SpitUnit Initialize maxDistance:100; velocity_up:100.0; velocity_down:100.0; acceleration:100000'		;															
fbSetAlarm[log_ID+1](
	InUse:=TRUE , 
	EventId:=log_ID+1 , 
	EventActive:=GVL_API.stSpitUnit.initialize, 
	EventClass:=Alm_EventClass.Event , 
	ToTheLogFile:=TRUE, 
	ToTheHistory:=TRUE , 
 );

 //home
AlarmActionArray[log_ID+2].AlarmMsg.EN	:=	'SpitUnit Home ';
fbSetAlarm[log_ID+2](
	InUse:=TRUE , 
	EventId:=log_ID+2 , 
	EventActive:=GVL_API.stSpitUnit.homeExe , 
	EventClass:=Alm_EventClass.Event , 
	ToTheLogFile:=TRUE, 
	ToTheHistory:=TRUE , 
 );
 
 //Move
AlarmActionArray[log_ID+3].AlarmMsg.EN	:=CONCAT('SpitUnit MoveAbsolute position:',
																	LREAL_TO_STRING(GVL_API.stSpitUnit.target_position));

fbSetAlarm[log_ID+3](
	InUse:=TRUE , 
	EventId:=log_ID+3 , 
	EventActive:=GVL_API.stSpitUnit.MoveAbsoluteExe , 
	EventClass:=Alm_EventClass.Event , 
	ToTheLogFile:=TRUE, 
	ToTheHistory:=TRUE , 
 );
 
//ERROR,log_ErrorEnum只能等于一个常数
CASE GVL_API.stSpitUnit.error_code  OF
0	:	log_ErrorEnum	:=	0	;
1	:	log_ErrorEnum	:=	1	;
2	:	log_ErrorEnum	:=	2	;
3	:	log_ErrorEnum	:=	3	;
4	:	log_ErrorEnum	:=	4	;
5	:	log_ErrorEnum	:=	5	;
6	:	log_ErrorEnum	:=	6	;
7	:	log_ErrorEnum	:=	7	;
8	:	log_ErrorEnum	:=	8	;
9	:	log_ErrorEnum	:=	9	;
666	:	log_ErrorEnum	:=	666	;

END_CASE

AlarmActionArray[log_ID+4].AlarmMsg.EN	:=CONCAT('SpitUnit Error: ',TO_STRING(log_ErrorEnum));
fbSetAlarm[log_ID+4](
	InUse:=TRUE , 
	EventId:=log_ID+4 , 
	EventActive:=GVL_API.stSpitUnit.error_code<>0 AND GVL_API.stSpitUnit.error_code<>666 , 
	EventClass:=Alm_EventClass.Alarm , 
	ToTheLogFile:=TRUE, 
	ToTheHistory:=TRUE , 
 );
 
//reset
AlarmActionArray[log_ID+5].AlarmMsg.EN	:=	'SpitUnit Reset ';
fbSetAlarm[log_ID+5](
	InUse:=TRUE , 
	EventId:=log_ID+5 , 
	EventActive:=GVL_API.stSpitUnit.setoff , 
	EventClass:=Alm_EventClass.Event , 
	ToTheLogFile:=TRUE, 
	ToTheHistory:=TRUE , 
 );
   //AXIX_ERRORID
 AlarmActionArray[log_ID+6].AlarmMsg.EN	:=CONCAT('SpitUnit Axis_ErrorID: ',
																		UDINT_TO_STRING(Axis[ID].Ref.Status.ErrorID));
fbSetAlarm[log_ID+6](
	InUse:=TRUE , 
	EventId:=log_ID+6 , 
	EventActive:=Axis[ID].Ref.Status.Error , 
	EventClass:=Alm_EventClass.Event , 
	ToTheLogFile:=TRUE, 
	ToTheHistory:=TRUE , 
 );
END_ACTION

ACTION ACT_Safety:
(*****************SAFETY******************************)
IF  GVL_API.stSpitUnit.state<>SpitUnitStateEnum.off AND GVL_API.stSpitUnit.state<>SpitUnitStateEnum.error THEN 
	IF GVL.Emstop_Button    THEN 	
		GVL_API.stSpitUnit.error_code:=SpitUnitErrorEnum.emergency_error;
		Axis[ID].aStop(stop_do:=TRUE);
		SysStep:=700;
	ELSIF GVL_API.stSpitUnit.state=SpitUnitStateEnum.moving AND Axis[ID].IO.snLimitP  THEN 
		GVL_API.stSpitUnit.error_code:=SpitUnitErrorEnum.trigger_limit;
		Axis[ID].aStop(stop_do:=TRUE);
		SysStep:=700;
	ELSIF  Axis[ID].mcReadStatus.ErrorID=18000 THEN 
		GVL_API.stAxis[ID].errorid:=Axis_XY_ErrorEnum.Drive_not_ready_for_operation;
		SysStep:=700;
	ELSIF  Axis[ID].mcReadStatus.ErrorID=17510 THEN 
		GVL_API.stAxis[ID].errorid:=Axis_XY_ErrorEnum.Invalid_IO_data_for_more_than_n_subsequent_NC_cycles_encoder;
		SysStep:=700;
	ELSIF  Axis[ID].mcReadStatus.ErrorID<>0 THEN 
		GVL_API.stAxis[ID].errorid:=Axis[ID].mcReadStatus.ErrorID;
		SysStep:=700;
	//ELSE 
	//	GVL_API.stAxis[ID].error:=Axis_XY_ErrorEnum.no_error;	
	//  SysStep:=700;
	END_IF
END_IF


(*****************AXIS_ERROR******************************)
GVL_API.stSpitUnit.AxisErrorId:=Axis[ID].Ref.Status.ErrorID;
END_ACTION

END_PROGRAM

// ---- GlobalTextList.TcGTLO
TEXTLIST GlobalTextList
  932 = '   CPU温度: \t%i oC'
  1595 = '   IP地址 1: \t%s'
  987 = '   IP地址 2: \t%s'
  1033 = '   TwinCAT等级: %s'
  940 = '   主板温度: \t%i oC'
  1598 = '   子网掩码1: \t%s'
  996 = '   子网掩码2: \t%s'
  1612 = '   程序名称: \t%s'
  1024 = '   程序日期: \t%s'
  1015 = '   程序版本: \t%s'
  949 = '   网卡1: \t%s'
  1873 = '  当前报警信息: %s'
  1042 = '  硬件日期: \t%s'
  1052 = '  系统NetId: \t%s'
  1602 = '  网卡2: \t%s'
  720 = '%.1f'
  18 = '%.2f'
  2502 = '%.2f '
  2635 = '%.2f  s '
  1353 = '%.2f min'
  1204 = '%.2f sec'
  3927 = '%.2f ℃'
  719 = '%d'
  2111 = '%D'
  2270 = '%i'
  233 = '%s'
  511 = '%s   '
  366 = '%t[ yyyy.MM.dd HH:mm:ss ]'
  1640 = '%u'
  711 = '+'
  945 = '-'
  1059 = '.2f'
  2147 = '1'
  2860 = '2'
  1039 = '3'
  2725 = '4'
  1993 = '5'
  335 = '6'
  2939 = '7'
  231 = '8'
  391 = '9'
  2431 = 'A:%d'
  504 = 'abs'
  219 = 'abs_pos:   %.4f'
  672 = 'acc:   %.1f'
  3164 = 'acc:   %.3f'
  1669 = 'ActEvent'
  2959 = 'Act_torque:   %.1f'
  1261 = 'Act_torque:   %d'
  300 = 'Admin'
  572 = 'AutoPos'
  314 = 'AXIS'
  276 = 'AxisErrorId:   %d'
  327 = 'Axis[3].IO.snLimitP'
  1004 = 'B'
  281 = 'back:%d'
  595 = 'back：%d'
  1935 = 'brake_timeout:   %.1f'
  1289 = 'brake_timeout:   %s'
  2246 = 'Break'
  252 = 'buzzer'
  1855 = 'BuzzerOff'
  2574 = 'BuzzerOn'
  16 = 'c'
  1003 = 'C'
  1770 = 'C1'
  1811 = 'C1:%s'
  1561 = 'C2'
  1217 = 'C2:%s'
  818 = 'CircPump1:   %.1f  V'
  97 = 'CircPump1_V:   %.1f'
  1581 = 'CircPump1_V:   %.1f  V'
  617 = 'CircPump2:   %.1f  V'
  2650 = 'CircPump2_V:   %.1f'
  3455 = 'circuit'
  1596 = 'circuit:   %.1f  V'
  2158 = 'CleanLog'
  1809 = 'CleeanLog'
  608 = 'Clutch'
  2055 = 'collision'
  2367 = 'collision_L'
  486 = 'collision_R'
  4009 = 'Com_err'
  612 = 'ConfigurePositions'
  2664 = 'continue:   %.1f'
  1025 = 'continue:   %.1f m'
  1013 = 'continue:   %.1f min'
  1814 = 'curing_started'
  2305 = 'curing_stopped'
  2288 = 'D:%.2f'
  1619 = 'dec:   %.1f'
  2770 = 'dec:   %.4f'
  491 = 'Delay_on:%.2f'
  1130 = 'Delay_on:%d'
  2748 = 'disable'
  977 = 'DisableBrake'
  1845 = 'down'
  2329 = 'dripping_allowed'
  1120 = 'DripTime_C'
  1322 = 'DripTime_W'
  273 = 'Drip_purge'
  1911 = 'duration:'
  1702 = 'EL1809_M_1'
  1711 = 'EL1809_M_2'
  1717 = 'EL1809_M_3'
  1402 = 'EL1809_S_1'
  1407 = 'EL1809_S_2'
  960 = 'EL1904_M_5'
  1352 = 'EL2809_M_1'
  1358 = 'EL2809_M_2'
  1364 = 'EL2809_M_3'
  1370 = 'EL2809_M_4'
  2278 = 'EL2809_S_1'
  338 = 'EL2904'
  503 = 'EL3064_M'
  2287 = 'EL4002_S'
  921 = 'Emstop'
  1784 = 'EM_STOP'
  2979 = 'en'
  305 = 'enable'
  2108 = 'EnableBrake'
  835 = 'end_pos:   %.4f'
  896 = 'Environment'
  2268 = 'error'
  2410 = 'Error'
  1342 = 'error:%s'
  2909 = 'errorID:%s'
  1315 = 'error_code'
  290 = 'EtherCAT'
  823 = 'EtherCAT Diag'
  2655 = 'Event'
  2759 = 'F'
  158 = 'F1'
  73 = 'F1:%s'
  420 = 'F2'
  2777 = 'F2:%s'
  759 = 'F:%s'
  701 = 'Fast SCAN'
  126 = 'FB_err'
  2071 = 'FB_SubTankFill_2[1].enable'
  170 = 'FB_SubTankFill_F[1].enable'
  190 = 'FB_SubTankFill_F[2].enable'
  2779 = 'FB_SubTankFill_W[1].enable'
  3384 = 'FB_SubTankFill_W[1].enable:   %.1f  V'
  1959 = 'FB_SubTankFill_W[2].enable'
  894 = 'FootPedal'
  796 = 'Frm0WcState'
  803 = 'Frm1WcState'
  810 = 'Frm2WcState'
  817 = 'Frm3WcState'
  3465 = 'has_dripped'
  994 = 'HMI手动设置能量'
  423 = 'home'
  479 = 'Home_Done'
  2903 = 'Homing'
  3603 = 'humidity_measured:'
  2267 = 'I:%.2f'
  991 = 'ini'
  1165 = 'Inide'
  1833 = 'Inied'
  26 = 'Initialize'
  3168 = 'initialized'
  1021 = 'Init_Done'
  1068 = 'InkSystem'
  2296 = 'INPUT1'
  764 = 'INPUT2'
  1247 = 'interlock'
  2832 = 'interlockMaintenanceUnitDoor'
  293 = 'interlockSpitUnitDoor'
  3241 = 'interlock_front_left'
  2634 = 'interlock_front_right'
  2445 = 'interlock_rear_left'
  1761 = 'interlock_rear_right'
  2648 = 'interShuttleDoor'
  415 = 'interva:   %.1f'
  3051 = 'interva:   %.1f m'
  3067 = 'IntervalTime_C'
  421 = 'IntervalTime_W'
  786 = 'IN_OUT1'
  787 = 'IN_OUT2'
  287 = 'IO1'
  288 = 'IO2'
  289 = 'IO3'
  1431 = 'is printing'
  270 = 'ISS'
  1475 = 'jerk:   %.1f'
  992 = 'jerk:   %.4f'
  1298 = 'K'
  1375 = 'K1'
  948 = 'K1:%s'
  368 = 'K2'
  1747 = 'K2:%s'
  1997 = 'LC'
  1216 = 'LC1'
  731 = 'lC1'
  28 = 'LC1:%s'
  947 = 'LC2'
  688 = 'LC2:%s'
  718 = 'LEFT:%d'
  1576 = 'LimitN'
  2784 = 'LimitP'
  3167 = 'limit_switch_bottom'
  2669 = 'limit_switch_left'
  433 = 'limit_switch_right'
  2805 = 'LM'
  2514 = 'LM1'
  246 = 'LM1:%s'
  1312 = 'LM2'
  882 = 'LM2:%s'
  1675 = 'LogEvent'
  3212 = 'L_Ahead_pos:%.1f'
  3105 = 'L_Delay_pos:%.1f'
  2077 = 'L_Lead_pos:%.1f'
  441 = 'L_Trailpos:%.1f'
  1132 = 'L_Trail_pos:%.1f'
  3669 = 'M'
  155 = 'M1'
  2169 = 'M1:%s'
  2235 = 'M2'
  119 = 'M2:%s'
  2925 = 'Main Tank Waste'
  3454 = 'Main Tank White '
  1815 = 'Main Tank White stirrer'
  271 = 'MaintenanceUnit'
  1663 = 'Max'
  2975 = 'max:%.1f kPa'
  700 = 'max:%.1f Pa'
  1156 = 'maxdis:   %.3f'
  484 = 'maxdis:   %.4f'
  2689 = 'MediaTransport'
  451 = 'min:%.1f kPa'
  181 = 'min:%.1f Pa'
  2051 = 'Monitor'
  2718 = 'MoveDown_do'
  1985 = 'MoveUp_do'
  225 = 'Move_Done'
  3247 = 'None'
  1659 = 'off'
  790 = 'off_pos:   %.4f'
  2473 = 'Operator'
  2065 = 'origin'
  1905 = 'Origin'
  1225 = 'OUTPUT1'
  1192 = 'OUTPUT2'
  914 = 'P'
  2028 = 'P1'
  590 = 'P1:%s'
  639 = 'P2'
  1354 = 'P2:%s'
  1082 = 'P:%.2f'
  3111 = 'period:'
  892 = 'PM1'
  123 = 'PM1:%s'
  673 = 'PM2'
  537 = 'PM2:%s'
  1859 = 'pos:   %.1f'
  988 = 'pos:   %.4f'
  535 = 'Power'
  1092 = 'PowerSettings'
  2933 = 'print_position:%d'
  43 = 'protect'
  3059 = 'PurgeTime_C'
  2601 = 'PurgeTime_W'
  1159 = 'PurgeValve7'
  3645 = 'range_pct:%.1f'
  1914 = 'rate:   %d'
  213 = 'rel'
  1927 = 'Remote'
  321 = 'Reset'
  1080 = 'rest'
  541 = 'rest_置位'
  1463 = 'RIGHT:%d'
  1657 = 'RTR'
  783 = 'Run'
  1310 = 'R_Ahead_pos:%.1f'
  2388 = 'R_Delay_pos:%.1f'
  2011 = 'R_Lead_pos:%.1f'
  2573 = 'R_Trail_pos:%.1f'
  965 = 'S1 Break'
  2220 = 'S1 En'
  632 = 'S1 Fr/Re'
  1240 = 'S1_Break'
  458 = 'S1_down'
  1835 = 'S1_En'
  2952 = 'S1_Fr/Re'
  895 = 'SaftyGuard'
  159 = 'sensor_down'
  2276 = 'sensor_up'
  1064 = 'Service'
  3198 = 'set:%.1f kPa'
  740 = 'set:%.1f Pa'
  42 = 'SetActivate'
  963 = 'setoff'
  106 = 'SetOff'
  216 = 'Setoff'
  1741 = 'SetReady'
  1051 = 'settings'
  2092 = 'settings_applide'
  591 = 'settings_applied'
  844 = 'SetVacuumOff'
  55 = 'SetVacuumOn'
  3246 = 'Set_torque:   %d'
  2735 = 'shuttle_crash_detector_left'
  336 = 'shuttle_crash_detector_right'
  67 = 'single_dual'
  571 = 'Slow SCAN'
  272 = 'SpitUnit'
  2157 = 'StartTension'
  351 = 'start_pos:   %.4f'
  791 = 'state'
  165 = 'state:%s'
  725 = 'step'
  716 = 'step:   %d'
  726 = 'stop'
  1655 = 'StopCuring'
  1526 = 'StopTension'
  1804 = 'stOutput.EL2904'
  2535 = 'SubTank'
  3481 = 'Swapping_Done'
  291 = 'SysInfo'
  1380 = 'System'
  294 = 'T'
  214 = 'TabVac'
  2503 = 'TEMP:%d'
  3314 = 'temp_measured: '
  2707 = 'tende'
  1695 = 'tension_mode'
  666 = 'tension_timeout:   %.1f'
  2135 = 'tension_timeout:   %s'
  732 = 'Ton.ET:%s'
  1278 = 'Ton_MoveDown'
  1243 = 'Ton_MoveUp'
  1531 = 'TwinSAFE_FBstop1_State'
  1283 = 'TwinSAFE_Group_State'
  361 = 'unidirection'
  1847 = 'unten'
  1254 = 'untension_timeout:   %.1f'
  2035 = 'untension_timeout:   %s'
  215 = 'UpDownSlot'
  1420 = 'uvEnd:   %.4f'
  1123 = 'UVLed'
  1516 = 'uvStart:   %.4f'
  559 = 'UV_LEFT'
  1242 = 'uv_power_leading:   %d'
  1384 = 'uv_power_trailing:   %d'
  1966 = 'UV_RIGHT'
  3339 = 'VacColorValve9'
  1532 = 'VacWhiteValve8'
  68 = 'velo'
  1710 = 'velo:   %.1f'
  534 = 'velo:   %.4f'
  2677 = 'velo_down:   %.3f'
  1621 = 'velo_up:   %.3f'
  312 = 'w'
  2893 = 'W'
  186 = 'W1'
  2693 = 'W1:%s'
  485 = 'W2'
  1122 = 'W2:%s'
  2964 = 'W3'
  2375 = 'W4'
  1129 = 'W:%d'
  2958 = 'Wast1:%s'
  422 = 'Wast2:%s'
  1329 = 'Waste'
  1860 = 'waste_level:%d'
  2790 = 'WL'
  704 = 'WR'
  1884 = 'X:%d'
  24 = 'Y'
  1258 = 'Y1'
  1103 = 'Y1:%s'
  2363 = 'Y2'
  506 = 'Y2:%s'
  435 = 'Y:%d'
  349 = 'Z'
  1885 = 'Z:%d'
  1633 = '修改'
  369 = '修改系统时间'
  881 = '关断超时:%.1f ms'
  3362 = '分'
  549 = '到达超时:%.1f ms'
  386 = '原点'
  2716 = '实际:%.1f Kpa'
  3474 = '实际:%.1f kPa'
  15 = '实际:%.1f Pa'
  352 = '年'
  363 = '当前时间'
  1183 = '手动设置能量'
  355 = '日'
  358 = '时'
  1636 = '月'
  350 = '正限位'
  957 = '电磁铁限位'
  931 = '读取'
  4013 = '负限位'
END_TEXTLIST

// ---- VISUs/base/title.TcVIS
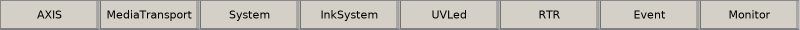
VISUALIZATION title  // 800x30
    Button (0,0 99x30), "AXIS"
        OnMouseDown: change screen: F1_AXIS
    Button (300,0 99x30), "InkSystem"
        OnMouseDown: change screen: F5_InkSystem
    Button (100,0 99x30), "MediaTransport"
        OnMouseDown: change screen: F3_MediaTransport
    Button (200,0 99x30), "System"
        OnMouseDown: change screen: F4_System
    Button (400,0 99x30), "UVLed"
        OnMouseDown: change screen: F6_UVLed
    Button (500,0 99x30), "RTR"
        OnMouseDown: change screen: F7_RTR
    Button (600,0 99x30), "Event"
        OnMouseDown: change screen: vis_arm
    Button (700,0 99x30), "Monitor"
        OnMouseDown: change screen: F99_Monitor
END_VISUALIZATION

// ---- VISUs/Components/IO_Components/F99_IO_IO.TcVIS
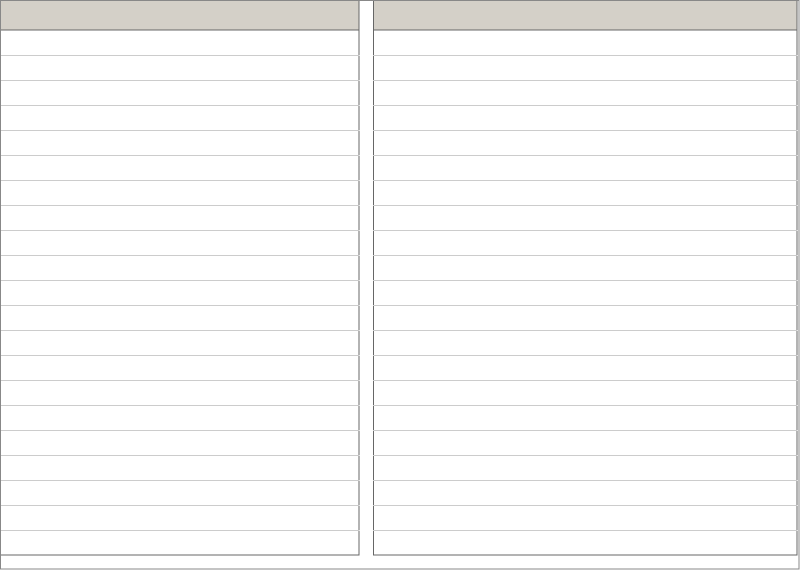
VISUALIZATION F99_IO_IO  // 800x570
    Table (0,0 359x555), data array: EL1809_M
        p1892666644: EL1809_M[2,INDEX]
        p338671338: EL1809_M[3,INDEX]
        p2685023577: EL1809_M[1,INDEX]
        Columns.Column.[0].Template: EL1809_M[1,INDEX]<>0
        Columns.Column.[1].Template: EL1809_M[2,INDEX]<>0
        Columns.Column.[2].Template: EL1809_M[3,INDEX]<>0
    Table (373,0 424x555), data array: EL2809_M
        p3854506369: EL2809_M[1,INDEX]
        p1892666644: EL2809_M[2,INDEX]
        p338671338: EL2809_M[3,INDEX]
        p2170511999: EL2809_M[4,INDEX]
        Columns.Column.[2].Template: EL2809_M[3,INDEX]<>0
        Columns.Column.[0].Template: EL2809_M[1,INDEX]<>0
        Columns.Column.[1].Template: EL2809_M[2,INDEX]<>0
        Columns.Column.[3].Template: EL2809_M[4,INDEX]<>0
END_VISUALIZATION

// ---- VISUs/Components/IO_Components/F99_IO_IO_1.TcVIS
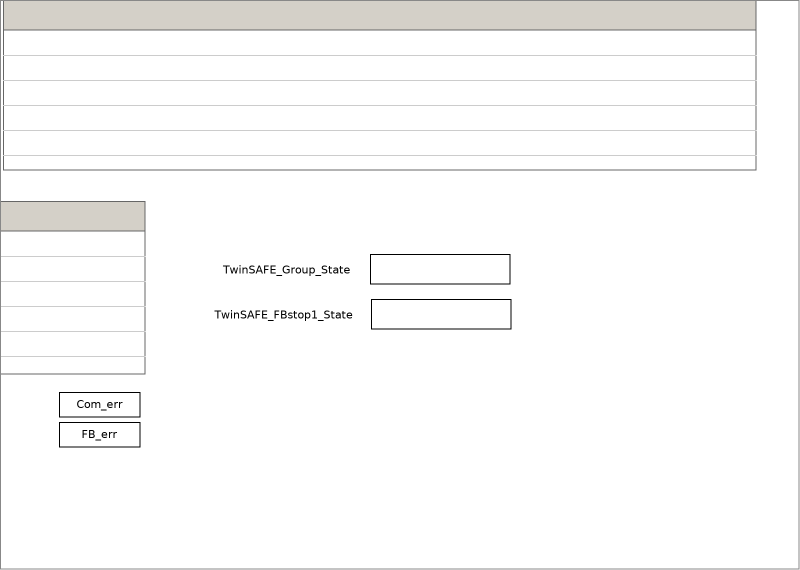
VISUALIZATION F99_IO_IO_1  // 800x570
    Table (3,0 753x170), data array: EL1904_M
        p3854506369: EL1904_M[1,INDEX]
        p1892666644: EL1904_M[2,INDEX]
        p338671338: EL1904_M[3,INDEX]
        p2170511999: EL1904_M[4,INDEX]
        p3723444502: EL1904_M[5,INDEX]
        Columns.Column.[0].Template: EL1904_M[1,INDEX]<>0
        Columns.Column.[1].Template: EL1904_M[2,INDEX]<>0
        Columns.Column.[2].Template: EL1904_M[3,INDEX]<>0
        Columns.Column.[3].Template: EL1904_M[4,INDEX]<>0
    Table (0,201 145x173), data array: EL2904
        p3854506369: EL2904[1,INDEX]
        p1892666644: EL2904[2,INDEX]
        p338671338: EL2904[3,INDEX]
        Columns.Column.[0].Template: EL2904[1,INDEX]<>0
    Rectangle (370,254 140x30), text list: 'TextList_TwinSAFE_Group_State', text index: P_TwinSAFE.TwinSAFE_Group_State
    Rectangle (371,299 140x30), text list: 'TextList_TwinSAFE_FB_ESTOP_State', text index: P_TwinSAFE.TwinSAFE_FBstop1_State
    Label (212,255 150x30), "TwinSAFE_Group_State"
    Label (209,300 150x30), "TwinSAFE_FBstop1_State"
    RoundedRectangle (59,422 81x25), "FB_err", colour toggle: P_TwinSAFE.FB_err
    RoundedRectangle (59,392 81x25), "Com_err", colour toggle: P_TwinSAFE.Com_err
END_VISUALIZATION

// ---- VISUs/Components/IO_Components/F99_IO_IO_2.TcVIS
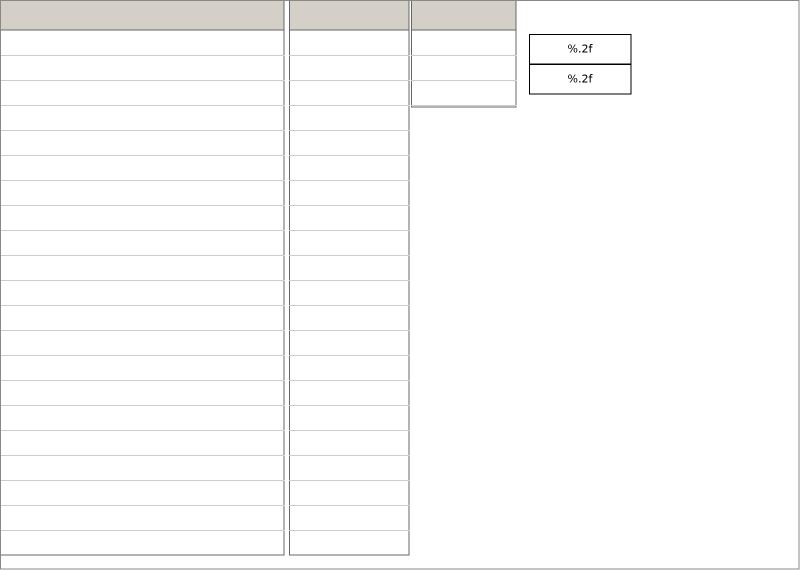
VISUALIZATION F99_IO_IO_2  // 800x570
    Table (0,0 284x555), data array: EL1809_S
        p3854506369: EL1809_S[1,INDEX]
        p1892666644: EL1809_S[2,INDEX]
        p338671338: EL1889_M[3,INDEX]
        Columns.Column.[1].Template: EL1809_S[2,INDEX]<>0
        Columns.Column.[0].Template: EL1809_S[1,INDEX]<>0
    Table (289,0 120x555), data array: EL2809_S
        p1892666644: EL2889_M[2,INDEX]
        p338671338: EL2889_M[3,INDEX]
        p2170511999: EL2889_M[4,INDEX]
        p3854506369: EL2809_S[1,INDEX]
        Columns.Column.[0].Template: EL2809_S[1,INDEX]<>0
    Table (411,0 105x107), data array: EL4002_S
        p3854506369: EL4002_S[INDEX]
    Rectangle (529,34 102x30), "%.2f", text variable: int_to_lreal(EL4002_S[1])/32767*10
    Rectangle (529,64 102x30), "%.2f", text variable: int_to_lreal(EL4002_S[2])/32767*10
END_VISUALIZATION

// ---- VISUs/Components/VIS_SubTank.TcVIS
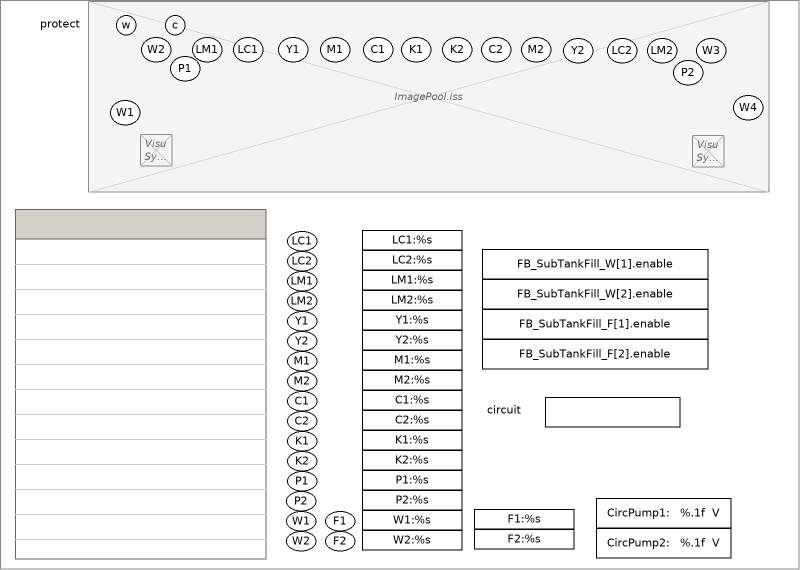
VISUALIZATION VIS_SubTank  // 800x570
    Image (88,1 681x191), image: ImagePool.iss
    Ellipse (116,15 20x20), "w", colour toggle: stInput.biProtectAirTankLevel_W
        toggle stInput.biProtectAirTankLevel_W
    Label (30,9 60x30), "protect"
    Ellipse (165,15 20x20), "c", colour toggle: stInput.biProtectAirTankLevel_C
        toggle stInput.biProtectAirTankLevel_C
    Group (110,37 653x130)
        Ellipse (0,63 30x25), "W1", colour toggle: stInput.biSubInkTankLevel[13]
            toggle stInput.biSubInkTankLevel[15]
        Ellipse (31,0 30x25), "W2", colour toggle: stInput.biSubInkTankLevel[14]
            toggle stInput.biSubInkTankLevel[16]
        Ellipse (123,0 30x25), "LC1", colour toggle: stInput.biSubInkTankLevel[1]
            toggle stInput.biSubInkTankLevel[11]
        Ellipse (82,0 30x25), "LM1", colour toggle: stInput.biSubInkTankLevel[3]
            toggle stInput.biSubInkTankLevel[9]
        Ellipse (168,0 30x25), "Y1", colour toggle: stInput.biSubInkTankLevel[5]
            toggle stInput.biSubInkTankLevel[1]
        Ellipse (210,0 30x25), "M1", colour toggle: stInput.biSubInkTankLevel[7]
            toggle stInput.biSubInkTankLevel[3]
        Ellipse (253,0 30x25), "C1", colour toggle: stInput.biSubInkTankLevel[9]
            toggle stInput.biSubInkTankLevel[5]
        Ellipse (291,0 30x25), "K1", colour toggle: stInput.biSubInkTankLevel[11]
            toggle stInput.biSubInkTankLevel[7]
        Ellipse (332,0 30x25), "K2", colour toggle: stInput.biSubInkTankLevel[12]
            toggle stInput.biSubInkTankLevel[8]
        Ellipse (371,0 30x25), "C2", colour toggle: stInput.biSubInkTankLevel[10]
            toggle stInput.biSubInkTankLevel[6]
        Ellipse (411,0 30x25), "M2", colour toggle: stInput.biSubInkTankLevel[8]
            toggle stInput.biSubInkTankLevel[4]
        Ellipse (453,1 30x25), "Y2", colour toggle: stInput.biSubInkTankLevel[6]
            toggle stInput.biSubInkTankLevel[2]
        Ellipse (537,1 30x25), "LM2", colour toggle: stInput.biSubInkTankLevel[4]
            toggle stInput.biSubInkTankLevel[10]
        Ellipse (497,1 30x25), "LC2", colour toggle: stInput.biSubInkTankLevel[2]
            toggle stInput.biSubInkTankLevel[12]
        Ellipse (586,1 30x25), "W3", colour toggle: stInput.biSubInkTankLevel[15]
            toggle stInput.biSubInkTankLevel[17]
        Ellipse (623,58 30x25), "W4", colour toggle: stInput.biSubInkTankLevel[16]
            toggle stInput.biSubInkTankLevel[18]
        Image (30,97 32x32), colour toggle: stOutput.bqSubCircPumpWorking[1], image: VisuSymbols.Symbols.ArrowQuarterLeftUp
        Image (582,98 32x32), colour toggle: stOutput.bqSubCircPumpWorking[2], image: VisuSymbols.Symbols.ArrowQuarterRightUp
        Ellipse (60,19 30x25), "P1", colour toggle: stInput.biSubInkTankLevel[17]
            toggle stInput.biSubInkTankLevel[13]
        Ellipse (563,23 30x25), "P2", colour toggle: stInput.biSubInkTankLevel[18]
            toggle stInput.biSubInkTankLevel[14]
    Ellipse (287,231 30x20), "LC1", colour toggle: stOutput.bqFillPumpWorking[1]
    Ellipse (287,271 30x20), "LM1", colour toggle: stOutput.bqFillPumpWorking[3]
    Ellipse (287,311 30x20), "Y1", colour toggle: stOutput.bqFillPumpWorking[5]
    Ellipse (287,351 30x20), "M1", colour toggle: stOutput.bqFillPumpWorking[7]
    Ellipse (287,391 30x20), "C1", colour toggle: stOutput.bqFillPumpWorking[9]
    Ellipse (287,251 30x20), "LC2", colour toggle: stOutput.bqFillPumpWorking[2]
    Ellipse (287,291 30x20), "LM2", colour toggle: stOutput.bqFillPumpWorking[4]
    Ellipse (287,331 30x20), "Y2", colour toggle: stOutput.bqFillPumpWorking[6]
    Ellipse (287,371 30x20), "M2", colour toggle: stOutput.bqFillPumpWorking[8]
    Ellipse (287,411 30x20), "C2", colour toggle: stOutput.bqFillPumpWorking[10]
    Ellipse (287,431 30x20), "K1", colour toggle: stOutput.bqFillPumpWorking[11]
    Ellipse (287,451 30x20), "K2", colour toggle: stOutput.bqFillPumpWorking[12]
    Ellipse (286,531 30x20), "W2", colour toggle: stOutput.bqFillPumpWorking[15]
    Ellipse (286,491 30x20), "P2", colour toggle: stOutput.bqFillPumpWorking[18]
    Ellipse (325,531 30x20), "F2", colour toggle: stOutput.bqFillPumpWorking[20]
    Ellipse (286,511 30x20), "W1", colour toggle: stOutput.bqFillPumpWorking[13]
    Ellipse (287,471 30x20), "P1", colour toggle: stOutput.bqFillPumpWorking[17]
    Ellipse (325,511 30x20), "F1", colour toggle: stOutput.bqFillPumpWorking[19]
    Rectangle (362,230 100x20), "LC1:%s", text variable: P_SubTank.FB_SubTankFill_C[1].inkFillTimeOutTon.ET
    Rectangle (362,270 100x20), "LM1:%s", text variable: P_SubTank.FB_SubTankFill_C[3].inkFillTimeOutTon.ET
    Rectangle (362,310 100x20), "Y1:%s", text variable: P_SubTank.FB_SubTankFill_C[5].inkFillTimeOutTon.ET
    Rectangle (362,350 100x20), "M1:%s", text variable: P_SubTank.FB_SubTankFill_C[7].inkFillTimeOutTon.ET
    Rectangle (362,390 100x20), "C1:%s", text variable: P_SubTank.FB_SubTankFill_C[9].inkFillTimeOutTon.ET
    Rectangle (362,430 100x20), "K1:%s", text variable: P_SubTank.FB_SubTankFill_C[11].inkFillTimeOutTon.ET
    Rectangle (362,510 100x20), "W1:%s", text variable: P_SubTank.FB_SubTankFill_W[1].inkFillTimeOutTon.ET
    Rectangle (362,470 100x20), "P1:%s", text variable: P_SubTank.FB_SubTankFill_P[1].inkFillTimeOutTon.ET
    Rectangle (474,509 100x20), "F1:%s", text variable: P_SubTank.FB_SubTankFill_F[1].inkFillTimeOutTon.ET
    Rectangle (362,250 100x20), "LC2:%s", text variable: P_SubTank.FB_SubTankFill_C[2].inkFillTimeOutTon.ET
    Rectangle (362,290 100x20), "LM2:%s", text variable: P_SubTank.FB_SubTankFill_C[4].inkFillTimeOutTon.ET
    Rectangle (362,330 100x20), "Y2:%s", text variable: P_SubTank.FB_SubTankFill_C[6].inkFillTimeOutTon.ET
    Rectangle (362,370 100x20), "M2:%s", text variable: P_SubTank.FB_SubTankFill_C[8].inkFillTimeOutTon.ET
    Rectangle (362,410 100x20), "C2:%s", text variable: P_SubTank.FB_SubTankFill_C[10].inkFillTimeOutTon.ET
    Rectangle (362,450 100x20), "K2:%s", text variable: P_SubTank.FB_SubTankFill_C[12].inkFillTimeOutTon.ET
    Rectangle (362,530 100x20), "W2:%s", text variable: P_SubTank.FB_SubTankFill_W[2].inkFillTimeOutTon.ET
    Rectangle (362,490 100x20), "P2:%s", text variable: P_SubTank.FB_SubTankFill_P[2].inkFillTimeOutTon.ET
    Rectangle (474,529 100x20), "F2:%s", text variable: P_SubTank.FB_SubTankFill_f[2].inkFillTimeOutTon.ET
    Rectangle (596,498 135x30), "CircPump1: %.1f V", text variable: HMI_CircPump1_V
        OnMouseDown: write HMI_CircPump1_V via Default, min 0, max 5
    Rectangle (596,528 135x30), "CircPump2: %.1f V", text variable: HMI_CircPump2_V
        OnMouseDown: write HMI_CircPump2_V via Default, min 0, max 5
    Rectangle (545,397 135x30), text list: 'TextList_SubTank_circuit', text index: SubTankInk_type
        OnMouseDown: write HMI_CircPump1_V via Default, min 0, max 5
    Rectangle (482,249 226x30), "FB_SubTankFill_W[1].enable", text variable: HMI_CircPump1_V, colour toggle: P_SubTank.FB_SubTankFill_W[1].enable
        OnMouseDown: write HMI_CircPump1_V via Default, min 0, max 5
    Rectangle (482,279 226x30), "FB_SubTankFill_W[2].enable", text variable: HMI_CircPump1_V, colour toggle: P_SubTank.FB_SubTankFill_W[2].enable
        OnMouseDown: write HMI_CircPump1_V via Default, min 0, max 5
    Rectangle (482,339 226x30), "FB_SubTankFill_F[2].enable", text variable: HMI_CircPump1_V, colour toggle: P_SubTank.FB_SubTankFill_F[2].enable
        OnMouseDown: write HMI_CircPump1_V via Default, min 0, max 5
    Rectangle (482,309 226x30), "FB_SubTankFill_F[1].enable", text variable: HMI_CircPump1_V, colour toggle: P_SubTank.FB_SubTankFill_F[1].enable
        OnMouseDown: write HMI_CircPump1_V via Default, min 0, max 5
    Label (474,395 60x30), "circuit"
    Table (15,209 251x350), data array: GVL_API.stSubTank
        p3854506369: GVL_API.stSubTank[INDEX].error_code
        p1892666644: GVL_API.stSubTank[INDEX].state
        p338671338: GVL_API.stSubTank[INDEX].Error
        p2170511999: GVL_API.stSubTank[INDEX].Setoff
        Columns.Column.[3].Template: toggle GVL_API.stSubTank[INDEX].Setoff
END_VISUALIZATION

// ---- VISUs/Components/VIS_RTR_2.TcVIS
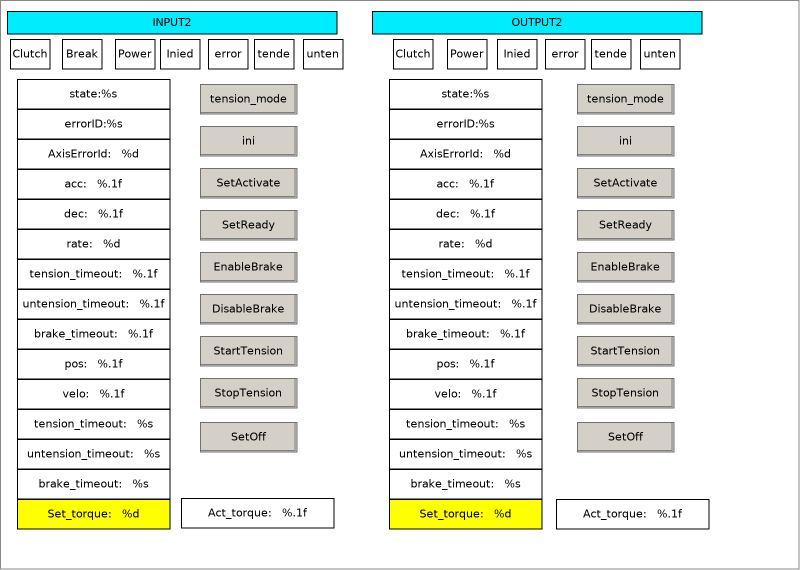
VISUALIZATION VIS_RTR_2  // 800x570
    RoundedRectangle (372,11 330x23), "OUTPUT2"
    RoundedRectangle (7,11 330x23), "INPUT2"
    Rectangle (17,79 153x30), "state:%s", colour toggle: GVL_API.stRoolToRool[3].state=100, text list: 'TextList_RTRstate', text index: GVL_API.stRoolToRool[3].state
    Rectangle (17,109 153x30), "errorID:%s", colour toggle: GVL_API.stRoolToRool[3].error_code<>0, text list: 'TextList_RTR_errorid', text index: GVL_API.stRoolToRool[3].error_code
    Rectangle (17,169 153x30), "acc: %.1f", text variable: GVL_API.stRoolToRool[3].acceleration
        OnMouseDown: write GVL_API.stRoolToRool[3].acceleration via Default
    Rectangle (17,199 153x30), "dec: %.1f", text variable: GVL_API.stRoolToRool[3].deceleration
        OnMouseDown: write GVL_API.stRoolToRool[3].deceleration via Default
    Rectangle (17,229 153x30), "rate: %d", text variable: GVL_API.stRoolToRool[3].rate
        OnMouseDown: write GVL_API.stRoolToRool[3].rate via Default
    Rectangle (17,259 153x30), "tension_timeout: %.1f", text variable: GVL_API.stRoolToRool[3].tension_timeout
        OnMouseDown: write GVL_API.stRoolToRool[3].tension_timeout via Default
    Rectangle (17,289 153x30), "untension_timeout: %.1f", text variable: GVL_API.stRoolToRool[3].untension_timeout
        OnMouseDown: write GVL_API.stRoolToRool[3].untension_timeout via Default
    Rectangle (17,319 153x30), "brake_timeout: %.1f", text variable: GVL_API.stRoolToRool[3].brake_timeout
        OnMouseDown: write GVL_API.stRoolToRool[3].brake_timeout via Default
    Rectangle (17,139 153x30), "AxisErrorId: %d", text variable: GVL_API.stRoolToRool[3].AxisErrorId
    RoundedRectangle (10,39 40x30), "Clutch", colour toggle: stOutput .bqCluthOut[3]
    RoundedRectangle (62,39 40x30), "Break", colour toggle: stOutput.bqBreakPower[3]
    Rectangle (389,79 153x30), "state:%s", colour toggle: GVL_API.stRoolToRool[4].state=100, text list: 'TextList_RTRstate', text index: GVL_API.stRoolToRool[4].state
    Rectangle (389,109 153x30), "errorID:%s", colour toggle: GVL_API.stRoolToRool[3].error_code<>0, text list: 'TextList_RTR_errorid', text index: GVL_API.stRoolToRool[4].error_code
    Rectangle (389,169 153x30), "acc: %.1f", text variable: GVL_API.stRoolToRool[4].acceleration
        OnMouseDown: write GVL_API.stRoolToRool[4].acceleration via Default
    Rectangle (389,199 153x30), "dec: %.1f", text variable: GVL_API.stRoolToRool[4].deceleration
        OnMouseDown: write GVL_API.stRoolToRool[4].deceleration via Default
    Rectangle (389,229 153x30), "rate: %d", text variable: GVL_API.stRoolToRool[4].rate
        OnMouseDown: write GVL_API.stRoolToRool[4].rate via Default
    Rectangle (389,259 153x30), "tension_timeout: %.1f", text variable: GVL_API.stRoolToRool[4].tension_timeout
        OnMouseDown: write GVL_API.stRoolToRool[4].tension_timeout via Default
    Rectangle (389,289 153x30), "untension_timeout: %.1f", text variable: GVL_API.stRoolToRool[4].untension_timeout
        OnMouseDown: write GVL_API.stRoolToRool[4].untension_timeout via Default
    Rectangle (389,319 153x30), "brake_timeout: %.1f", text variable: GVL_API.stRoolToRool[4].brake_timeout
        OnMouseDown: write GVL_API.stRoolToRool[4].brake_timeout via Default
    Rectangle (389,139 153x30), "AxisErrorId: %d", text variable: GVL_API.stRoolToRool[4].AxisErrorId
    RoundedRectangle (393,39 40x30), "Clutch", colour toggle: stOutput .bqCluthOut[4]
    Button (200,126 97x30), "ini", colour toggle: GVL_API.stRoolToRool[3].Initialize
        toggle GVL_API.stRoolToRool[3].Initialize
    Button (200,84 97x30), "tension_mode", colour toggle: GVL_API.stRoolToRool[3].tension_mode
        toggle GVL_API.stRoolToRool[3].tension_mode
    Button (200,168 97x30), "SetActivate", colour toggle: GVL_API.stRoolToRool[3].SetActivate
        toggle GVL_API.stRoolToRool[3].SetActivate
    Button (200,294 97x30), "DisableBrake", colour toggle: GVL_API.stRoolToRool[3].DisableBrake
        toggle GVL_API.stRoolToRool[3].DisableBrake
    Button (200,210 97x30), "SetReady", colour toggle: GVL_API.stRoolToRool[3].SetReady
        toggle GVL_API.stRoolToRool[3].SetReady
    Button (200,252 97x30), "EnableBrake", colour toggle: GVL_API.stRoolToRool[3].EnableBrake
        toggle GVL_API.stRoolToRool[3].EnableBrake
    Button (200,336 97x30), "StartTension", colour toggle: GVL_API.stRoolToRool[3].StartTension
        toggle GVL_API.stRoolToRool[3].StartTension
    Button (200,378 97x30), "StopTension", colour toggle: GVL_API.stRoolToRool[3].StopTension
        toggle GVL_API.stRoolToRool[3].StopTension
    Button (200,422 97x30), "SetOff", colour toggle: GVL_API.stRoolToRool[3].SetOff
        toggle GVL_API.stRoolToRool[3].SetOff
    Button (577,126 97x30), "ini", colour toggle: GVL_API.stRoolToRool[4].Initialize
        toggle GVL_API.stRoolToRool[4].Initialize
    Button (577,84 97x30), "tension_mode", colour toggle: GVL_API.stRoolToRool[4].tension_mode
        toggle GVL_API.stRoolToRool[4].tension_mode
    Button (577,168 97x30), "SetActivate", colour toggle: GVL_API.stRoolToRool[4].SetActivate
        toggle GVL_API.stRoolToRool[4].SetActivate
    Button (577,294 97x30), "DisableBrake", colour toggle: GVL_API.stRoolToRool[4].DisableBrake
        toggle GVL_API.stRoolToRool[4].DisableBrake
    Button (577,210 97x30), "SetReady", colour toggle: GVL_API.stRoolToRool[4].SetReady
        toggle GVL_API.stRoolToRool[4].SetReady
    Button (577,252 97x30), "EnableBrake", colour toggle: GVL_API.stRoolToRool[4].EnableBrake
        toggle GVL_API.stRoolToRool[4].EnableBrake
    Button (577,336 97x30), "StartTension", colour toggle: GVL_API.stRoolToRool[4].StartTension
        toggle GVL_API.stRoolToRool[4].StartTension
    Button (577,378 97x30), "StopTension", colour toggle: GVL_API.stRoolToRool[4].StopTension
        toggle GVL_API.stRoolToRool[4].StopTension
    Button (577,422 97x30), "SetOff", colour toggle: GVL_API.stRoolToRool[4].SetOff
        toggle GVL_API.stRoolToRool[4].SetOff
    RoundedRectangle (447,39 40x30), "Power", colour toggle: P_RollToRoll.FB_RoolToRool[4].REF.Status.ControlLoopClosed
    RoundedRectangle (115,39 40x30), "Power", colour toggle: P_RollToRoll.FB_RoolToRool[3].REF.Status.ControlLoopClosed
    Rectangle (17,349 153x30), "pos: %.1f", text variable: P_RollToRoll.FB_RoolToRool[3].REF.NcToPlc.ActPos
        OnMouseDown: write GVL_API.stRoolToRool[1].brake_timeout via Default
    Rectangle (17,379 153x30), "velo: %.1f", text variable: P_RollToRoll.FB_RoolToRool[3].REF.NcToPlc.ActVelo
        OnMouseDown: write GVL_API.stRoolToRool[1].brake_timeout via Default
    Rectangle (389,349 153x30), "pos: %.1f", text variable: P_RollToRoll.FB_RoolToRool[4].REF.NcToPlc.ActPos
        OnMouseDown: write GVL_API.stRoolToRool[1].brake_timeout via Default
    Rectangle (389,379 153x30), "velo: %.1f", text variable: P_RollToRoll.FB_RoolToRool[4].REF.NcToPlc.ActVelo
        OnMouseDown: write GVL_API.stRoolToRool[1].brake_timeout via Default
    Rectangle (17,409 153x30), "tension_timeout: %s", text variable: P_RollToRoll.FB_RoolToRool[3].tension_ton.ET
    Rectangle (17,439 153x30), "untension_timeout: %s", text variable: P_RollToRoll.FB_RoolToRool[3].untension_ton.ET
    Rectangle (17,469 153x30), "brake_timeout: %s", text variable: P_RollToRoll.FB_RoolToRool[3].enbreak_ton.ET
    Rectangle (389,409 153x30), "tension_timeout: %s", text variable: P_RollToRoll.FB_RoolToRool[4].tension_ton.ET
    Rectangle (389,439 153x30), "untension_timeout: %s", text variable: P_RollToRoll.FB_RoolToRool[4].untension_ton.ET
    Rectangle (389,469 153x30), "brake_timeout: %s", text variable: P_RollToRoll.FB_RoolToRool[4].enbreak_ton.ET
    Rectangle (17,499 153x30), "Set_torque: %d", text variable: HMI_RTR_set_Torque[3]
        OnMouseDown: write HMI_RTR_set_Torque[3] via Default, min 0, max 100
    Rectangle (389,499 153x30), "Set_torque: %d", text variable: HMI_RTR_set_Torque[4]
        OnMouseDown: write HMI_RTR_set_Torque[4] via Default, min 0, max 100
    Rectangle (181,498 153x30), "Act_torque: %.1f", text variable: P_RollToRoll.FB_RoolToRool[3].REF.NcToPlc.ActTorque
    Rectangle (556,499 153x30), "Act_torque: %.1f", text variable: P_RollToRoll.FB_RoolToRool[4].REF.NcToPlc.ActTorque
    RoundedRectangle (160,39 40x30), "Inied", colour toggle: P_RollToRoll.FB_RoolToRool[3].Initialized
    RoundedRectangle (208,39 40x30), "error", colour toggle: P_RollToRoll.FB_RoolToRool[3].error
    RoundedRectangle (254,39 40x30), "tende", colour toggle: P_RollToRoll.FB_RoolToRool[3].tensioned
    RoundedRectangle (303,39 40x30), "unten", colour toggle: P_RollToRoll.FB_RoolToRool[3].untensioned
    RoundedRectangle (497,39 40x30), "Inied", colour toggle: P_RollToRoll.FB_RoolToRool[4].Initialized
    RoundedRectangle (545,39 40x30), "error", colour toggle: P_RollToRoll.FB_RoolToRool[4].error
    RoundedRectangle (591,39 40x30), "tende", colour toggle: P_RollToRoll.FB_RoolToRool[4].tensioned
    RoundedRectangle (640,39 40x30), "unten", colour toggle: P_RollToRoll.FB_RoolToRool[4].untensioned
END_VISUALIZATION

// ---- VISUs/Components/VIS_SpitUnit.TcVIS
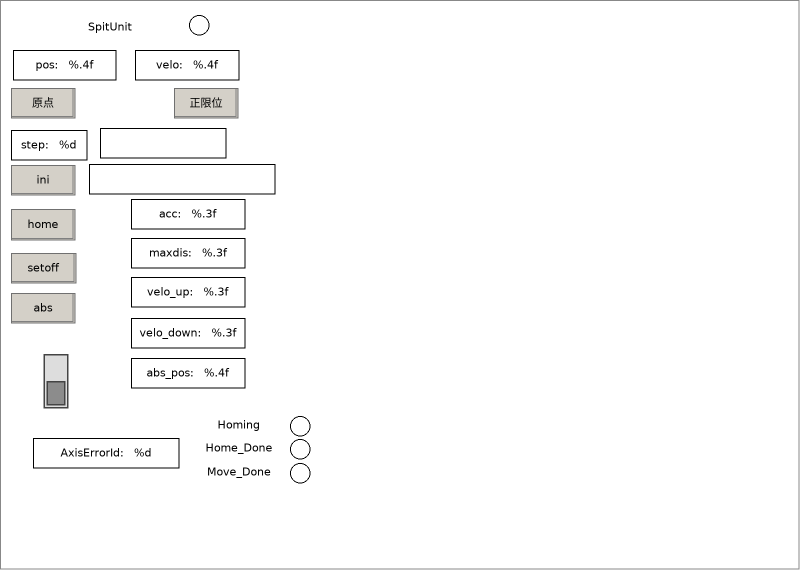
VISUALIZATION VIS_SpitUnit  // 800x570
    Button (11,209 64x31), "home", colour toggle: GVL_API.stSpitUnit.HomeExe
        toggle GVL_API.stSpitUnit.HomeExe
    Button (11,88 64x30), "原点", colour toggle: Axis[4].IO.snHome
        toggle Axis[4].IO.snHome
    Button (174,88 64x30), "正限位", colour toggle: Axis[4].IO.snLimitP
        toggle Axis[4].IO.snLimitP
    Rectangle (13,50 103x30), "pos: %.4f", text variable: Axis[4].Ref.NcToPlc.ActPos
    Rectangle (135,50 104x30), "velo: %.4f", text variable: Axis[4].Ref.NcToPlc.ActVelo
    Ellipse (189,15 20x20), colour toggle: Axis[4].Ref.Status.ControlLoopClosed
    Button (11,293 64x30), "abs", colour toggle: GVL_API.stSpitUnit.MoveAbsoluteExe
        toggle GVL_API.stSpitUnit.MoveAbsoluteExe
    Button (11,165 64x30), "ini", colour toggle: GVL_API.stSpitUnit.Initialize
        toggle GVL_API.stSpitUnit.Initialize
    Rectangle (131,358 114x30), "abs_pos: %.4f", text variable: GVL_API.stSpitUnit.target_position
        OnMouseDown: write GVL_API.stSpitUnit.target_position via Default
    Rectangle (131,277 114x30), "velo_up: %.3f", text variable: GVL_API.stSpitUnit.moving_speed_up
        OnMouseDown: write GVL_API.stSpitUnit.moving_speed_up via Default
    Rectangle (11,130 76x30), "step: %d", text variable: P_SpitUnit.SysStep
        OnMouseDown: write P_SpitUnit.SysStep via Default
    Button (11,253 65x30), "setoff", colour toggle: GVL_API.stSpitUnit.SetOff
        toggle GVL_API.stSpitUnit.SetOff
    Rectangle (100,128 126x30), text list: 'TextListSpitUnitState', text index: GVL_API.stSpitUnit.state
    Rectangle (89,164 186x30), text list: 'TextListSpitUnitErrorid', text index: GVL_API.stSpitUnit.error_code
    Label (70,12 80x30), "SpitUnit"
    Rectangle (33,438 146x30), "AxisErrorId: %d", text variable: GVL_API.stSpitUnit.AxisErrorId
    Rectangle (131,238 114x30), "maxdis: %.3f", text variable: GVL_API.stSpitUnit.spindle_length
        OnMouseDown: write GVL_API.stSpitUnit.spindle_length via Default
    Rectangle (131,199 114x30), "acc: %.3f", text variable: GVL_API.stSpitUnit.acceleration
        OnMouseDown: write GVL_API.stSpitUnit.acceleration via Default
    Rectangle (131,318 114x30), "velo_down: %.3f", text variable: GVL_API.stSpitUnit.moving_speed_down
        OnMouseDown: write GVL_API.stSpitUnit.moving_speed_down via Default
    Label (199,433 80x30), "Home_Done"
    Ellipse (290,439 20x20), colour toggle: GVL_API.stSpitUnit.Home_Done
    Label (199,457 80x30), "Move_Done"
    Ellipse (290,463 20x20), colour toggle: GVL_API.stSpitUnit.Move_Done
    DipSwitch (29,354 54x54), variable: GVL.HMI_btEmstop, behaviour: TOGGLE, style: Switch-DipSwitch-Gray
    Label (199,410 80x30), "Homing"
    Ellipse (290,416 20x20), colour toggle: GVL_API.stSpitUnit.Homing
END_VISUALIZATION

// ---- VISUs/Components/VIS_TabVac.TcVIS
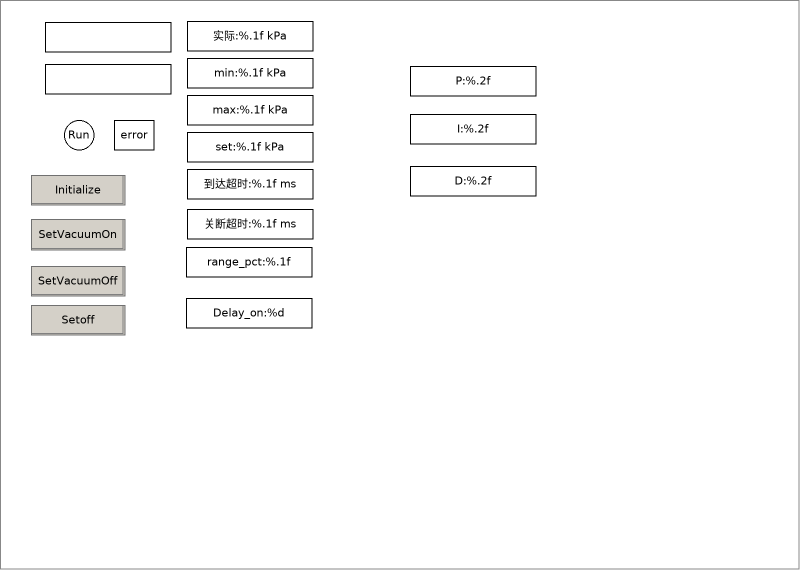
VISUALIZATION VIS_TabVac  // 800x570
    Rectangle (45,22 126x30), text list: 'TextList_tabvac_state', text index: GVL_API.stTableVacuum[1].state
    Button (31,175 94x30), "Initialize", colour toggle: GVL_API.stTableVacuum[1].Initialize
        toggle GVL_API.stTableVacuum[1].Initialize
    Button (31,219 94x31), "SetVacuumOn", colour toggle: GVL_API.stTableVacuum[1].SetVacuumOn
        toggle GVL_API.stTableVacuum[1].SetVacuumOn
        OnMouseDown: execute { GVL_API.stAxis[1].homingvelocity:=100; }
    Button (31,266 94x30), "SetVacuumOff", colour toggle: GVL_API.stTableVacuum[1].SetVacuumOff
        toggle GVL_API.stTableVacuum[1].SetVacuumOff
    Button (31,305 94x30), "Setoff", colour toggle: GVL_API.stTableVacuum[1].Setoff
        toggle GVL_API.stTableVacuum[1].Setoff
    Rectangle (187,21 126x30), "实际:%.1f kPa", text variable: GVL_API.stTableVacuum[1].vacuum_measured
        OnMouseDown: write GVL_API.stTableVacuum[1].vacuum_measured via Default
    Rectangle (187,58 126x30), "min:%.1f kPa", text variable: GVL_API.stTableVacuum[1].vacuum_min
        OnMouseDown: write GVL_API.stTableVacuum[1].vacuum_min via Default
    Rectangle (187,95 126x30), "max:%.1f kPa", text variable: GVL_API.stTableVacuum[1].vacuum_max
        OnMouseDown: write GVL_API.stTableVacuum[1].vacuum_max via Default
    Rectangle (187,169 126x30), "到达超时:%.1f ms", text variable: GVL_API.stTableVacuum[1].vacuum_timeout
        OnMouseDown: write GVL_API.stTableVacuum[1].vacuum_timeout via Default
    Rectangle (187,209 126x30), "关断超时:%.1f ms", text variable: GVL_API.stTableVacuum[1].vacuum_off_timeout
        OnMouseDown: write GVL_API.stTableVacuum[1].vacuum_off_timeout via Default
    Ellipse (64,120 30x30), "Run", colour toggle: stOutput.bqVacRun[1]
    Rectangle (187,132 126x30), "set:%.1f kPa", text variable: GVL_API.stTableVacuum[1].setpoint
        OnMouseDown: write GVL_API.stTableVacuum[1].setpoint via Default
    Rectangle (186,247 126x30), "range_pct:%.1f", text variable: GVL_API.stTableVacuum[1].setpoint_range_pct
        OnMouseDown: write GVL_API.stTableVacuum[1].setpoint_range_pct via Default
    Rectangle (45,64 126x30), text list: 'TextList_tabvac_errorid', text index: GVL_API.stTableVacuum[1].error_code
    Rectangle (410,66 126x30), "P:%.2f", text variable: GVL_API.stTableVacuum[1].ctrlP
        OnMouseDown: write GVL_API.stTableVacuum[1].ctrlP via Default
    Rectangle (410,114 126x30), "I:%.2f", text variable: GVL_API.stTableVacuum[1].ctrlI
        OnMouseDown: write GVL_API.stTableVacuum[1].ctrlI via Default
    Rectangle (410,166 126x30), "D:%.2f", text variable: GVL_API.stTableVacuum[1].ctrlD
        OnMouseDown: write GVL_API.stTableVacuum[1].ctrlD via Default
    RoundedRectangle (114,120 40x30), "error", colour toggle: GVL_API.stTableVacuum[1].Error
    Rectangle (186,298 126x30), "Delay_on:%d", text variable: HMI_Vac_dely_on
        OnMouseDown: write HMI_Vac_dely_on via Default, min 0
END_VISUALIZATION

